KUKA KRL program: EPS_2_251806_MH49A_A_20260213065148.src

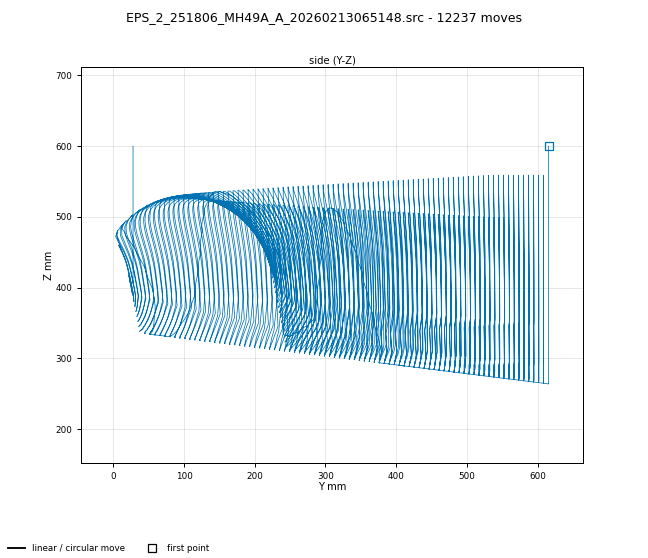
[picture p0: tool path of EPS_2_251806_MH49A_A_20260213065148.src, 12237 of 12239 moves have a stored position in this frame; points joined in program order, loops and branches not executed]
&ACCESS RVP
&REL 4
&COMMENT QRS 19112012
&PARAM EDITMASK = *
DEF PART()
EXT BAS (BAS_COMMAND :IN,REAL :IN )
INT I
BAS (#INITMOV,0 )

;KUKA QRS Post kuka4.cps  Date:22-06-2017 !

File_ID=3036

QRS_PRE_INIT()

;Init var - Until changes are made in qrs_pre_init
Outlet_Square_prg=0
Inlet_1_Square_prg=0
Inlet_2_Square_prg=0
Inlet_3_Square_prg=0
Inlet_4_Square_prg=0
Inlet_5_Square_prg=0

Outlet_1={X 0.000, Y 535.490, Z 458.500, B 0.000, E1 0.000 }
Inlet_1={X 0.000, Y 539.770, Z 398.500, B 0.000, E1 242.000 }
Outlet_1_type=201
Inlet_1_type=201
;QRS#1=Sidecore dimensions
;QRS#2=200-8" PVC SDR 35
;QRS#3=200-8" PVC SDR 35
;QRS#4=
;QRS#5=
;QRS#6=
;QRS#7=
;QRS#8=
;QRS#9=12-08 PSX
;QRS#10=12-08 PSX
;QRS#11=
;QRS#12=
;QRS#13=
;QRS#14=
;QRS#15=
;QRS#16=1220x127x838 2,75'
;QRS#17=EPS Height
;QRS#18=559
;QRS#19=*
;QRS#20= UPDATED VERSION 22-06-2017
;QRS#21=*
Outlet_Square=0100
Inlet_1_Square=0100
Inlet_2_Square=0
Inlet_3_Square=0
Inlet_4_Square=0
Inlet_5_Square=0
Mill_Square=1
Outlet_Square_Prg=204
Inlet_1_Square_prg=204

QRS_INIT()

$ADVANCE=5

; T1
PTP {E1 173.582,E2 173.582}
PTP {X 0,Y 615.48,A -85,B 0,C 180,E1 173.582,E2 173.582,E3 0,E4 0,E5 0,E6 0}
QRS_SPEED_INIT()
LIN {X 0,Y 615.48,Z 600,A -85,B 0,C 180,E1 173.582,E2 173.582,E3 0,E4 0,E5 0,E6 0} C_VEL
LIN {X 0,Y 615.48,Z 273.871,A -85,B 0,C 180,E1 173.582,E2 173.582} C_VEL
LIN {X 0,Y 615.48,Z 265.699,A -85,B 0,C 180,E1 173.582,E2 173.582} C_VEL
LIN {X 0,Y 615.469,Z 263.699,A -85,B 0,C 180,E1 173.396,E2 173.396} C_VEL
LIN {X 0,Y 615.482,Z 263.691,A -85,B 0,C 180,E1 170.801,E2 170.801} C_VEL
LIN {X 0,Y 615.433,Z 263.694,A -85,B 0,C 180,E1 168.138,E2 168.138} C_VEL
LIN {X 0,Y 615.433,Z 263.694,A -85,B 0,C 180,E1 166.069,E2 166.069} C_VEL
LIN {X 0,Y 615.451,Z 263.697,A -85,B 0,C 180,E1 163.565,E2 163.565} C_VEL
LIN {X 0,Y 615.479,Z 263.689,A -85,B 0,C 180,E1 160.662,E2 160.662} C_VEL
LIN {X 0,Y 615.473,Z 263.689,A -85,B 0,C 180,E1 158.568,E2 158.568} C_VEL
LIN {X 0,Y 615.439,Z 263.693,A -85,B 0,C 180,E1 155.991,E2 155.991} C_VEL
LIN {X 0,Y 615.452,Z 263.696,A -85,B 0,C 180,E1 153.555,E2 153.555} C_VEL
LIN {X 0,Y 615.483,Z 263.688,A -85,B 0,C 180,E1 150.594,E2 150.594} C_VEL
LIN {X 0,Y 615.462,Z 263.688,A -85,B 0,C 180,E1 148.314,E2 148.314} C_VEL
LIN {X 0,Y 615.443,Z 263.692,A -85,B 0,C 180,E1 145.976,E2 145.976} C_VEL
LIN {X 0,Y 615.453,Z 263.695,A -85,B 0,C 180,E1 143.573,E2 143.573} C_VEL
LIN {X 0,Y 615.495,Z 263.696,A -85,B 0,C 180,E1 140.932,E2 140.932} C_VEL
LIN {X 0,Y 615.496,Z 263.684,A -85,B 0,C 180,E1 138.527,E2 138.527} C_VEL
LIN {X 0,Y 615.449,Z 263.691,A -85,B 0,C 180,E1 135.847,E2 135.847} C_VEL
LIN {X 0,Y 615.487,Z 263.703,A -85,B 0,C 180,E1 133.048,E2 133.048} C_VEL
LIN {X 0,Y 615.465,Z 263.687,A -85,B 0,C 180,E1 130.087,E2 130.087} C_VEL
LIN {X 0,Y 615.462,Z 263.687,A -85,B 0,C 180,E1 128.01,E2 128.01} C_VEL
LIN {X 0,Y 615.456,Z 263.692,A -85,B 0,C 180,E1 125.615,E2 125.615} C_VEL
LIN {X 0,Y 615.472,Z 263.698,A -85,B 0,C 180,E1 123.235,E2 123.235} C_VEL
LIN {X 0,Y 615.488,Z 263.699,A -85,B 0,C 180,E1 120.917,E2 120.917} C_VEL
LIN {X 0,Y 615.466,Z 263.687,A -85,B 0,C 180,E1 117.914,E2 117.914} C_VEL
LIN {X 0,Y 615.461,Z 263.692,A -85,B 0,C 180,E1 115.565,E2 115.565} C_VEL
LIN {X 0,Y 615.487,Z 263.698,A -85,B 0,C 180,E1 112.843,E2 112.843} C_VEL
LIN {X 0,Y 615.481,Z 263.683,A -85,B 0,C 180,E1 110.032,E2 110.032} C_VEL
LIN {X 0,Y 615.473,Z 263.695,A -85,B 0,C 180,E1 107.27,E2 107.27} C_VEL
LIN {X 0,Y 615.485,Z 263.69,A -85,B 0,C 180,E1 104.549,E2 104.549} C_VEL
LIN {X 0,Y 615.477,Z 263.684,A -85,B 0,C 180,E1 101.861,E2 101.861} C_VEL
LIN {X 0,Y 615.477,Z 263.696,A -85,B 0,C 180,E1 99.199,E2 99.199} C_VEL
LIN {X 0,Y 615.483,Z 263.691,A -85,B 0,C 180,E1 96.557,E2 96.557} C_VEL
LIN {X 0,Y 615.485,Z 263.682,A -85,B 0,C 180,E1 93.929,E2 93.929} C_VEL
LIN {X 0,Y 615.474,Z 263.693,A -85,B 0,C 180,E1 91.31,E2 91.31} C_VEL
LIN {X 0,Y 615.485,Z 263.696,A -85,B 0,C 180,E1 88.693,E2 88.693} C_VEL
LIN {X 0,Y 615.487,Z 263.682,A -85,B 0,C 180,E1 86.073,E2 86.073} C_VEL
LIN {X 0,Y 615.475,Z 263.689,A -85,B 0,C 180,E1 83.429,E2 83.429} C_VEL
LIN {X 0,Y 615.49,Z 263.699,A -85,B 0,C 180,E1 80.803,E2 80.803} C_VEL
LIN {X 0,Y 615.481,Z 263.685,A -85,B 0,C 180,E1 78.141,E2 78.141} C_VEL
LIN {X 0,Y 615.478,Z 263.687,A -85,B 0,C 180,E1 75.453,E2 75.453} C_VEL
LIN {X 0,Y 615.488,Z 263.698,A -85,B 0,C 180,E1 72.732,E2 72.732} C_VEL
LIN {X 0,Y 615.484,Z 263.683,A -85,B 0,C 180,E1 69.97,E2 69.97} C_VEL
LIN {X 0,Y 615.482,Z 263.693,A -85,B 0,C 180,E1 67.159,E2 67.159} C_VEL
LIN {X 0,Y 615.474,Z 263.693,A -85,B 0,C 180,E1 64.433,E2 64.433} C_VEL
LIN {X 0,Y 615.473,Z 263.687,A -85,B 0,C 180,E1 62.088,E2 62.088} C_VEL
LIN {X 0,Y 615.483,Z 263.683,A -85,B 0,C 180,E1 59.844,E2 59.844} C_VEL
LIN {X 0,Y 615.494,Z 263.682,A -85,B 0,C 180,E1 57.548,E2 57.548} C_VEL
LIN {X 0,Y 615.484,Z 263.69,A -85,B 0,C 180,E1 55.19,E2 55.19} C_VEL
LIN {X 0,Y 615.491,Z 263.701,A -85,B 0,C 180,E1 52.764,E2 52.764} C_VEL
LIN {X 0,Y 615.47,Z 263.686,A -85,B 0,C 180,E1 49.912,E2 49.912} C_VEL
LIN {X 0,Y 615.487,Z 263.682,A -85,B 0,C 180,E1 47.654,E2 47.654} C_VEL
LIN {X 0,Y 615.489,Z 263.799,A -85,B 0,C 180,E1 45.291,E2 45.291} C_VEL
LIN {X 0,Y 615.45,Z 278.087,A -85,B 0,C 180,E1 42.705,E2 42.705} C_VEL
LIN {X 0,Y 615.463,Z 288.652,A -85,B 0,C 180,E1 40.808,E2 40.808} C_VEL
LIN {X 0,Y 615.487,Z 395.253,A -85,B 0,C 180,E1 39.537,E2 39.537} C_VEL
LIN {X 0,Y 615.489,Z 408.573,A -85,B 0,C 180,E1 39.239,E2 39.239} C_VEL
LIN {X 0,Y 615.487,Z 421.763,A -85,B 0,C 180,E1 38.799,E2 38.799} C_VEL
LIN {X 0,Y 615.467,Z 433.203,A -85,B 0,C 180,E1 38.278,E2 38.278} C_VEL
LIN {X 0,Y 615.479,Z 444.346,A -85,B 0,C 180,E1 37.629,E2 37.629} C_VEL
LIN {X 0,Y 615.495,Z 455.472,A -85,B 0,C 180,E1 36.816,E2 36.816} C_VEL
LIN {X 0,Y 615.497,Z 464.537,A -85,B 0,C 180,E1 35.989,E2 35.989} C_VEL
LIN {X 0,Y 615.496,Z 473.253,A -85,B 0,C 180,E1 35.014,E2 35.014} C_VEL
LIN {X 0,Y 615.496,Z 480.397,A -85,B 0,C 180,E1 34.021,E2 34.021} C_VEL
LIN {X 0,Y 615.496,Z 484.99,A -85,B 0,C 180,E1 33.235,E2 33.235} C_VEL
LIN {X 0,Y 615.493,Z 490.657,A -85,B 0,C 180,E1 32.013,E2 32.013} C_VEL
LIN {X 0,Y 615.497,Z 494.308,A -85,B 0,C 180,E1 30.919,E2 30.919} C_VEL
LIN {X 0,Y 615.496,Z 496.791,A -85,B 0,C 180,E1 29.808,E2 29.808} C_VEL
LIN {X 0,Y 615.497,Z 498.269,A -85,B 0,C 180,E1 28.465,E2 28.465} C_VEL
LIN {X 0,Y 615.496,Z 498.086,A -85,B 0,C 180,E1 27.176,E2 27.176} C_VEL
LIN {X 0,Y 615.494,Z 497.341,A -85,B 0,C 180,E1 26.443,E2 26.443} C_VEL
LIN {X 0,Y 615.495,Z 495.782,A -85,B 0,C 180,E1 25.585,E2 25.585} C_VEL
LIN {X 0,Y 615.495,Z 493.234,A -85,B 0,C 180,E1 24.631,E2 24.631} C_VEL
LIN {X 0,Y 615.496,Z 489.236,A -85,B 0,C 180,E1 23.556,E2 23.556} C_VEL
LIN {X 0,Y 615.496,Z 484.603,A -85,B 0,C 180,E1 22.604,E2 22.604} C_VEL
LIN {X 0,Y 615.495,Z 478.501,A -85,B 0,C 180,E1 21.607,E2 21.607} C_VEL
LIN {X 0,Y 615.497,Z 470.633,A -85,B 0,C 180,E1 20.578,E2 20.578} C_VEL
LIN {X 0,Y 615.497,Z 462.118,A -85,B 0,C 180,E1 19.684,E2 19.684} C_VEL
LIN {X 0,Y 615.498,Z 451.961,A -85,B 0,C 180,E1 18.818,E2 18.818} C_VEL
LIN {X 0,Y 615.464,Z 441.937,A -85,B 0,C 180,E1 18.125,E2 18.125} C_VEL
LIN {X 0,Y 615.471,Z 431.12,A -85,B 0,C 180,E1 17.528,E2 17.528} C_VEL
LIN {X 0,Y 615.474,Z 418.019,A -85,B 0,C 180,E1 16.971,E2 16.971} C_VEL
LIN {X 0,Y 615.451,Z 405.553,A -85,B 0,C 180,E1 16.587,E2 16.587} C_VEL
LIN {X 0,Y 615.45,Z 392.084,A -85,B 0,C 180,E1 16.325,E2 16.325} C_VEL
LIN {X 0,Y 615.493,Z 288.624,A -85,B 0,C 180,E1 15.098,E2 15.098} C_VEL
LIN {X 0,Y 615.482,Z 274.331,A -85,B 0,C 180,E1 12.53,E2 12.53} C_VEL
LIN {X 0,Y 615.427,Z 263.699,A -85,B 0,C 180,E1 10.576,E2 10.576} C_VEL
LIN {X 0,Y 615.425,Z 263.699,A -85,B 0,C 180,E1 8.537,E2 8.537} C_VEL
LIN {X 0,Y 615.426,Z 263.699,A -85,B 0,C 180,E1 6.557,E2 6.557} C_VEL
LIN {X 0,Y 615.435,Z 263.698,A -85,B 0,C 180,E1 4.585,E2 4.585} C_VEL
LIN {X 0,Y 615.44,Z 263.698,A -85,B 0,C 180,E1 2.618,E2 2.618} C_VEL
LIN {X 0,Y 615.412,Z 263.699,A -85,B 0,C 180,E1 0,E2 0} C_VEL
LIN {X 0,Y 615.451,Z 263.699,A -85,B 0,C 180,E1 -2.618,E2 -2.618} C_VEL
LIN {X 0,Y 615.468,Z 263.697,A -85,B 0,C 180,E1 -5.242,E2 -5.242} C_VEL
LIN {X 0,Y 615.417,Z 263.698,A -85,B 0,C 180,E1 -7.877,E2 -7.877} C_VEL
LIN {X 0,Y 615.419,Z 263.697,A -85,B 0,C 180,E1 -9.864,E2 -9.864} C_VEL
LIN {X 0,Y 615.42,Z 263.697,A -85,B 0,C 180,E1 -11.862,E2 -11.862} C_VEL
LIN {X 0,Y 615.419,Z 263.697,A -85,B 0,C 180,E1 -13.935,E2 -13.935} C_VEL
LIN {X 0,Y 615.421,Z 263.697,A -85,B 0,C 180,E1 -15.907,E2 -15.907} C_VEL
LIN {X 0,Y 615.421,Z 263.697,A -85,B 0,C 180,E1 -17.959,E2 -17.959} C_VEL
LIN {X 0,Y 615.418,Z 263.697,A -85,B 0,C 180,E1 -20.035,E2 -20.035} C_VEL
LIN {X 0,Y 615.422,Z 263.698,A -85,B 0,C 180,E1 -22.348,E2 -22.348} C_VEL
LIN {X 0,Y 615.481,Z 263.7,A -85,B 0,C 180,E1 -24.992,E2 -24.992} C_VEL
LIN {X 0,Y 615.486,Z 263.701,A -85,B 0,C 180,E1 -27.178,E2 -27.178} C_VEL
LIN {X 0,Y 615.423,Z 263.696,A -85,B 0,C 180,E1 -30.164,E2 -30.164} C_VEL
LIN {X 0,Y 615.427,Z 263.697,A -85,B 0,C 180,E1 -32.461,E2 -32.461} C_VEL
LIN {X 0,Y 615.45,Z 263.699,A -85,B 0,C 180,E1 -34.818,E2 -34.818} C_VEL
LIN {X 0,Y 615.496,Z 263.699,A -85,B 0,C 180,E1 -37.242,E2 -37.242} C_VEL
LIN {X 0,Y 615.431,Z 263.695,A -85,B 0,C 180,E1 -40.091,E2 -40.091} C_VEL
LIN {X 0,Y 615.425,Z 263.696,A -85,B 0,C 180,E1 -42.359,E2 -42.359} C_VEL
LIN {X 0,Y 615.431,Z 263.694,A -85,B 0,C 180,E1 -44.155,E2 -44.155} C_VEL
LIN {X 0,Y 615.457,Z 263.698,A -85,B 0,C 180,E1 -46.956,E2 -46.956} C_VEL
LIN {X 0,Y 615.453,Z 263.692,A -85,B 0,C 180,E1 -49.915,E2 -49.915} C_VEL
LIN {X 0,Y 615.448,Z 263.693,A -85,B 0,C 180,E1 -51.993,E2 -51.993} C_VEL
LIN {X 0,Y 615.43,Z 263.694,A -85,B 0,C 180,E1 -54.386,E2 -54.386} C_VEL
LIN {X 0,Y 615.434,Z 263.697,A -85,B 0,C 180,E1 -56.766,E2 -56.766} C_VEL
LIN {X 0,Y 615.463,Z 263.698,A -85,B 0,C 180,E1 -59.084,E2 -59.084} C_VEL
LIN {X 0,Y 615.451,Z 263.692,A -85,B 0,C 180,E1 -62.087,E2 -62.087} C_VEL
LIN {X 0,Y 615.434,Z 263.694,A -85,B 0,C 180,E1 -64.442,E2 -64.442} C_VEL
LIN {X 0,Y 615.435,Z 263.73,A -85,B 0,C 180,E1 -66.69,E2 -66.69} C_VEL
LIN {X 0,Y 615.481,Z 283.686,A -85,B 0,C 180,E1 -69.272,E2 -69.272} C_VEL
LIN {X 0,Y 615.476,Z 305.498,A -85,B 0,C 180,E1 -72.046,E2 -72.046} C_VEL
LIN {X 0,Y 615.49,Z 327.283,A -85,B 0,C 180,E1 -74.777,E2 -74.777} C_VEL
LIN {X 0,Y 615.45,Z 346.155,A -85,B 0,C 180,E1 -77.115,E2 -77.115} C_VEL
LIN {X 0,Y 615.457,Z 454.961,A -85,B 0,C 180,E1 -78.412,E2 -78.412} C_VEL
LIN {X 0,Y 615.456,Z 467.431,A -85,B 0,C 180,E1 -78.683,E2 -78.683} C_VEL
LIN {X 0,Y 615.483,Z 480.691,A -85,B 0,C 180,E1 -79.116,E2 -79.116} C_VEL
LIN {X 0,Y 615.49,Z 492.517,A -85,B 0,C 180,E1 -79.642,E2 -79.642} C_VEL
LIN {X 0,Y 615.488,Z 504.026,A -85,B 0,C 180,E1 -80.306,E2 -80.306} C_VEL
LIN {X 0,Y 615.499,Z 514.366,A -85,B 0,C 180,E1 -81.052,E2 -81.052} C_VEL
LIN {X 0,Y 615.497,Z 522.832,A -85,B 0,C 180,E1 -81.796,E2 -81.796} C_VEL
LIN {X 0,Y 615.497,Z 531.98,A -85,B 0,C 180,E1 -82.786,E2 -82.786} C_VEL
LIN {X 0,Y 615.498,Z 539.326,A -85,B 0,C 180,E1 -83.774,E2 -83.774} C_VEL
LIN {X 0,Y 615.498,Z 545.213,A -85,B 0,C 180,E1 -84.76,E2 -84.76} C_VEL
LIN {X 0,Y 615.494,Z 549.858,A -85,B 0,C 180,E1 -85.745,E2 -85.745} C_VEL
LIN {X 0,Y 615.494,Z 553.403,A -85,B 0,C 180,E1 -86.728,E2 -86.728} C_VEL
LIN {X 0,Y 615.497,Z 555.236,A -85,B 0,C 180,E1 -87.383,E2 -87.383} C_VEL
LIN {X 0,Y 615.498,Z 556.61,A -85,B 0,C 180,E1 -88.038,E2 -88.038} C_VEL
LIN {X 0,Y 615.496,Z 558.174,A -85,B 0,C 180,E1 -89.347,E2 -89.347} C_VEL
LIN {X 0,Y 615.494,Z 558.389,A -85,B 0,C 180,E1 -90.001,E2 -90.001} C_VEL
LIN {X 0,Y 615.495,Z 557.579,A -85,B 0,C 180,E1 -91.309,E2 -91.309} C_VEL
LIN {X 0,Y 615.498,Z 556.606,A -85,B 0,C 180,E1 -91.964,E2 -91.964} C_VEL
LIN {X 0,Y 615.497,Z 555.231,A -85,B 0,C 180,E1 -92.619,E2 -92.619} C_VEL
LIN {X 0,Y 615.496,Z 552.347,A -85,B 0,C 180,E1 -93.601,E2 -93.601} C_VEL
LIN {X 0,Y 615.498,Z 548.439,A -85,B 0,C 180,E1 -94.585,E2 -94.585} C_VEL
LIN {X 0,Y 615.499,Z 543.402,A -85,B 0,C 180,E1 -95.57,E2 -95.57} C_VEL
LIN {X 0,Y 615.497,Z 536.87,A -85,B 0,C 180,E1 -96.583,E2 -96.583} C_VEL
LIN {X 0,Y 615.497,Z 529.13,A -85,B 0,C 180,E1 -97.546,E2 -97.546} C_VEL
LIN {X 0,Y 615.498,Z 521.043,A -85,B 0,C 180,E1 -98.371,E2 -98.371} C_VEL
LIN {X 0,Y 615.499,Z 511.166,A -85,B 0,C 180,E1 -99.199,E2 -99.199} C_VEL
LIN {X 0,Y 615.489,Z 499.98,A -85,B 0,C 180,E1 -99.945,E2 -99.945} C_VEL
LIN {X 0,Y 615.489,Z 489.022,A -85,B 0,C 180,E1 -100.527,E2 -100.527} C_VEL
LIN {X 0,Y 615.469,Z 476.532,A -85,B 0,C 180,E1 -101.039,E2 -101.039} C_VEL
LIN {X 0,Y 615.454,Z 464.076,A -85,B 0,C 180,E1 -101.402,E2 -101.402} C_VEL
LIN {X 0,Y 615.459,Z 450.483,A -85,B 0,C 180,E1 -101.652,E2 -101.652} C_VEL
LIN {X 0,Y 615.449,Z 346.138,A -85,B 0,C 180,E1 -102.887,E2 -102.887} C_VEL
LIN {X 0,Y 615.48,Z 325.904,A -85,B 0,C 180,E1 -105.395,E2 -105.395} C_VEL
LIN {X 0,Y 615.485,Z 304.214,A -85,B 0,C 180,E1 -108.116,E2 -108.116} C_VEL
LIN {X 0,Y 615.485,Z 282.304,A -85,B 0,C 180,E1 -110.905,E2 -110.905} C_VEL
LIN {X 0,Y 615.435,Z 263.712,A -85,B 0,C 180,E1 -113.312,E2 -113.312} C_VEL
LIN {X 0,Y 615.44,Z 263.693,A -85,B 0,C 180,E1 -115.716,E2 -115.716} C_VEL
LIN {X 0,Y 615.48,Z 263.702,A -85,B 0,C 180,E1 -118.656,E2 -118.656} C_VEL
LIN {X 0,Y 615.444,Z 263.698,A -85,B 0,C 180,E1 -121.079,E2 -121.079} C_VEL
LIN {X 0,Y 615.434,Z 263.697,A -85,B 0,C 180,E1 -123.237,E2 -123.237} C_VEL
LIN {X 0,Y 615.427,Z 263.695,A -85,B 0,C 180,E1 -125.617,E2 -125.617} C_VEL
LIN {X 0,Y 615.452,Z 263.694,A -85,B 0,C 180,E1 -128.068,E2 -128.068} C_VEL
LIN {X 0,Y 615.442,Z 263.698,A -85,B 0,C 180,E1 -131.089,E2 -131.089} C_VEL
LIN {X 0,Y 615.43,Z 263.698,A -85,B 0,C 180,E1 -133.246,E2 -133.246} C_VEL
LIN {X 0,Y 615.436,Z 263.696,A -85,B 0,C 180,E1 -136.003,E2 -136.003} C_VEL
LIN {X 0,Y 615.464,Z 263.699,A -85,B 0,C 180,E1 -138.903,E2 -138.903} C_VEL
LIN {X 0,Y 615.44,Z 263.7,A -85,B 0,C 180,E1 -141.092,E2 -141.092} C_VEL
LIN {X 0,Y 615.414,Z 263.699,A -85,B 0,C 180,E1 -143.57,E2 -143.57} C_VEL
LIN {X 0,Y 615.468,Z 263.699,A -85,B 0,C 180,E1 -146.462,E2 -146.462} C_VEL
LIN {X 0,Y 615.444,Z 263.7,A -85,B 0,C 180,E1 -149.078,E2 -149.078} C_VEL
LIN {X 0,Y 615.41,Z 263.7,A -85,B 0,C 180,E1 -151.555,E2 -151.555} C_VEL
LIN {X 0,Y 615.409,Z 263.7,A -85,B 0,C 180,E1 -153.552,E2 -153.552} C_VEL
LIN {X 0,Y 615.414,Z 263.7,A -85,B 0,C 180,E1 -155.997,E2 -155.997} C_VEL
LIN {X 0,Y 615.471,Z 263.7,A -85,B 0,C 180,E1 -158.567,E2 -158.567} C_VEL
LIN {X 0,Y 615.424,Z 263.699,A -85,B 0,C 180,E1 -161.399,E2 -161.399} C_VEL
LIN {X 0,Y 615.416,Z 263.698,A -85,B 0,C 180,E1 -163.575,E2 -163.575} C_VEL
LIN {X 0,Y 615.424,Z 263.698,A -85,B 0,C 180,E1 -165.449,E2 -165.449} C_VEL
LIN {X 0,Y 615.426,Z 263.697,A -85,B 0,C 180,E1 -167.468,E2 -167.468} C_VEL
LIN {X 0,Y 615.428,Z 263.697,A -85,B 0,C 180,E1 -169.472,E2 -169.472} C_VEL
LIN {X 0,Y 615.431,Z 263.696,A -85,B 0,C 180,E1 -171.462,E2 -171.462} C_VEL
LIN {X 0,Y 615.432,Z 263.697,A -85,B 0,C 180,E1 -173.442,E2 -173.442} C_VEL
LIN {X 0,Y 615.44,Z 263.695,A -85,B 0,C 180,E1 -175.415,E2 -175.415} C_VEL
LIN {X 0,Y 615.446,Z 263.695,A -85,B 0,C 180,E1 -177.382,E2 -177.382} C_VEL
LIN {X 0,Y 615.452,Z 263.694,A -85,B 0,C 180,E1 -179.345,E2 -179.345} C_VEL
LIN {X 0,Y 615.425,Z 263.696,A -85,B 0,C 180,E1 -181.963,E2 -181.963} C_VEL
LIN {X 0,Y 615.467,Z 263.699,A -85,B 0,C 180,E1 -184.584,E2 -184.584} C_VEL
LIN {X 0,Y 615.469,Z 263.699,A -85,B 0,C 180,E1 -186.604,E2 -186.604} C_VEL
LIN {X 0,Y 614.804,Z 263.839,A -85,B 0,C 180,E1 -187.15,E2 -187.15} C_VEL
LIN {X 0,Y 611.979,Z 264.248,A -85,B 0,C 180,E1 -188.036,E2 -188.036} C_VEL
LIN {X 0,Y 609.581,Z 264.561,A -85,B 0,C 180,E1 -188.749,E2 -188.749} C_VEL
LIN {X 0,Y 608.531,Z 264.681,A -85,B 0,C 180,E1 -189.298,E2 -189.298} C_VEL
LIN {X 0,Y 608.434,Z 264.691,A -85,B 0,C 180,E1 -189.484,E2 -189.484} C_VEL
LIN {X 0,Y 608.415,Z 264.692,A -85,B 0,C 180,E1 -192,E2 -192} C_VEL
LIN {X 0,Y 608.454,Z 264.696,A -85,B 0,C 180,E1 -194.721,E2 -194.721} C_VEL
LIN {X 0,Y 608.433,Z 264.691,A -85,B 0,C 180,E1 -197.477,E2 -197.477} C_VEL
LIN {X 0,Y 608.427,Z 264.691,A -85,B 0,C 180,E1 -199.571,E2 -199.571} C_VEL
LIN {X 0,Y 608.434,Z 264.693,A -85,B 0,C 180,E1 -202.406,E2 -202.406} C_VEL
LIN {X 0,Y 608.443,Z 264.692,A -85,B 0,C 180,E1 -205.301,E2 -205.301} C_VEL
LIN {X 0,Y 608.428,Z 264.692,A -85,B 0,C 180,E1 -207.519,E2 -207.519} C_VEL
LIN {X 0,Y 608.43,Z 264.69,A -85,B 0,C 180,E1 -209.973,E2 -209.973} C_VEL
LIN {X 0,Y 608.43,Z 264.694,A -85,B 0,C 180,E1 -212.525,E2 -212.525} C_VEL
LIN {X 0,Y 608.436,Z 264.694,A -85,B 0,C 180,E1 -215.278,E2 -215.278} C_VEL
LIN {X 0,Y 608.445,Z 264.688,A -85,B 0,C 180,E1 -217.748,E2 -217.748} C_VEL
LIN {X 0,Y 608.422,Z 264.693,A -85,B 0,C 180,E1 -220.331,E2 -220.331} C_VEL
LIN {X 0,Y 608.456,Z 264.698,A -85,B 0,C 180,E1 -222.959,E2 -222.959} C_VEL
LIN {X 0,Y 608.437,Z 264.689,A -85,B 0,C 180,E1 -225.737,E2 -225.737} C_VEL
LIN {X 0,Y 608.442,Z 264.688,A -85,B 0,C 180,E1 -227.941,E2 -227.941} C_VEL
LIN {X 0,Y 608.465,Z 264.692,A -85,B 0,C 180,E1 -230.702,E2 -230.702} C_VEL
LIN {X 0,Y 608.465,Z 264.695,A -85,B 0,C 180,E1 -233.089,E2 -233.089} C_VEL
LIN {X 0,Y 608.466,Z 264.688,A -85,B 0,C 180,E1 -235.533,E2 -235.533} C_VEL
LIN {X 0,Y 608.461,Z 264.686,A -85,B 0,C 180,E1 -237.908,E2 -237.908} C_VEL
LIN {X 0,Y 608.446,Z 264.688,A -85,B 0,C 180,E1 -240.221,E2 -240.221} C_VEL
LIN {X 0,Y 608.475,Z 264.691,A -85,B 0,C 180,E1 -242.793,E2 -242.793} C_VEL
LIN {X 0,Y 608.472,Z 264.685,A -85,B 0,C 180,E1 -245.848,E2 -245.848} C_VEL
LIN {X 0,Y 608.456,Z 264.688,A -85,B 0,C 180,E1 -248.309,E2 -248.309} C_VEL
LIN {X 0,Y 608.451,Z 264.697,A -85,B 0,C 180,E1 -251.131,E2 -251.131} C_VEL
LIN {X 0,Y 608.455,Z 264.687,A -85,B 0,C 180,E1 -253.907,E2 -253.907} C_VEL
LIN {X 0,Y 608.451,Z 264.691,A -85,B 0,C 180,E1 -256.644,E2 -256.644} C_VEL
LIN {X 0,Y 608.463,Z 264.691,A -85,B 0,C 180,E1 -259.35,E2 -259.35} C_VEL
LIN {X 0,Y 608.474,Z 264.684,A -85,B 0,C 180,E1 -262.033,E2 -262.033} C_VEL
LIN {X 0,Y 608.456,Z 264.691,A -85,B 0,C 180,E1 -264.698,E2 -264.698} C_VEL
LIN {X 0,Y 608.474,Z 264.69,A -85,B 0,C 180,E1 -267.351,E2 -267.351} C_VEL
LIN {X 0,Y 608.477,Z 264.684,A -85,B 0,C 180,E1 -269.999,E2 -269.999} C_VEL
LIN {X 0,Y 608.466,Z 264.689,A -85,B 0,C 180,E1 -272.647,E2 -272.647} C_VEL
LIN {X 0,Y 608.466,Z 264.693,A -85,B 0,C 180,E1 -275.3,E2 -275.3} C_VEL
LIN {X 0,Y 608.474,Z 264.684,A -85,B 0,C 180,E1 -277.965,E2 -277.965} C_VEL
LIN {X 0,Y 608.458,Z 264.689,A -85,B 0,C 180,E1 -280.648,E2 -280.648} C_VEL
LIN {X 0,Y 608.465,Z 264.692,A -85,B 0,C 180,E1 -283.354,E2 -283.354} C_VEL
LIN {X 0,Y 608.456,Z 264.687,A -85,B 0,C 180,E1 -286.091,E2 -286.091} C_VEL
LIN {X 0,Y 608.447,Z 264.694,A -85,B 0,C 180,E1 -288.867,E2 -288.867} C_VEL
LIN {X 0,Y 608.464,Z 264.688,A -85,B 0,C 180,E1 -291.688,E2 -291.688} C_VEL
LIN {X 0,Y 608.451,Z 264.689,A -85,B 0,C 180,E1 -294.567,E2 -294.567} C_VEL
LIN {X 0,Y 608.476,Z 264.695,A -85,B 0,C 180,E1 -297.208,E2 -297.208} C_VEL
LIN {X 0,Y 608.454,Z 264.687,A -85,B 0,C 180,E1 -299.97,E2 -299.97} C_VEL
LIN {X 0,Y 608.463,Z 264.687,A -85,B 0,C 180,E1 -302.523,E2 -302.523} C_VEL
LIN {X 0,Y 608.434,Z 264.699,A -85,B 0,C 180,E1 -305.273,E2 -305.273} C_VEL
LIN {X 0,Y 608.457,Z 264.689,A -85,B 0,C 180,E1 -307.741,E2 -307.741} C_VEL
LIN {X 0,Y 608.447,Z 264.688,A -85,B 0,C 180,E1 -310.329,E2 -310.329} C_VEL
LIN {X 0,Y 608.48,Z 264.694,A -85,B 0,C 180,E1 -313.31,E2 -313.31} C_VEL
LIN {X 0,Y 608.502,Z 264.835,A -85,B 0,C 180,E1 -314.674,E2 -314.674} C_VEL
LIN {X 0,Y 608.432,Z 279.669,A -85,B 0,C 180,E1 -317.38,E2 -317.38} C_VEL
LIN {X 0,Y 608.439,Z 288.884,A -85,B 0,C 180,E1 -319.046,E2 -319.046} C_VEL
LIN {X 0,Y 608.552,Z 395.169,A -85,B 0,C 180,E1 -320.326,E2 -320.326} C_VEL
LIN {X 0,Y 608.547,Z 408.611,A -85,B 0,C 180,E1 -320.628,E2 -320.628} C_VEL
LIN {X 0,Y 608.517,Z 421.099,A -85,B 0,C 180,E1 -321.045,E2 -321.045} C_VEL
LIN {X 0,Y 608.487,Z 431.65,A -85,B 0,C 180,E1 -321.515,E2 -321.515} C_VEL
LIN {X 0,Y 608.464,Z 442.542,A -85,B 0,C 180,E1 -322.128,E2 -322.128} C_VEL
LIN {X 0,Y 608.491,Z 452.552,A -85,B 0,C 180,E1 -322.83,E2 -322.83} C_VEL
LIN {X 0,Y 608.474,Z 462.7,A -85,B 0,C 180,E1 -323.705,E2 -323.705} C_VEL
LIN {X 0,Y 608.449,Z 470.445,A -85,B 0,C 180,E1 -324.52,E2 -324.52} C_VEL
LIN {X 0,Y 608.459,Z 478.293,A -85,B 0,C 180,E1 -325.53,E2 -325.53} C_VEL
LIN {X 0,Y 608.432,Z 484.497,A -85,B 0,C 180,E1 -326.526,E2 -326.526} C_VEL
LIN {X 0,Y 608.43,Z 489.222,A -85,B 0,C 180,E1 -327.471,E2 -327.471} C_VEL
LIN {X 0,Y 608.447,Z 493.912,A -85,B 0,C 180,E1 -328.721,E2 -328.721} C_VEL
LIN {X 0,Y 608.446,Z 495.945,A -85,B 0,C 180,E1 -329.454,E2 -329.454} C_VEL
LIN {X 0,Y 608.442,Z 497.468,A -85,B 0,C 180,E1 -330.22,E2 -330.22} C_VEL
LIN {X 0,Y 608.423,Z 498.778,A -85,B 0,C 180,E1 -331.376,E2 -331.376} C_VEL
LIN {X 0,Y 608.427,Z 498.726,A -85,B 0,C 180,E1 -332.789,E2 -332.789} C_VEL
LIN {X 0,Y 608.416,Z 497.313,A -85,B 0,C 180,E1 -333.964,E2 -333.964} C_VEL
LIN {X 0,Y 608.428,Z 494.822,A -85,B 0,C 180,E1 -335.064,E2 -335.064} C_VEL
LIN {X 0,Y 608.437,Z 491.173,A -85,B 0,C 180,E1 -336.154,E2 -336.154} C_VEL
LIN {X 0,Y 608.456,Z 486.303,A -85,B 0,C 180,E1 -337.231,E2 -337.231} C_VEL
LIN {X 0,Y 608.458,Z 479.982,A -85,B 0,C 180,E1 -338.308,E2 -338.308} C_VEL
LIN {X 0,Y 608.462,Z 472.656,A -85,B 0,C 180,E1 -339.305,E2 -339.305} C_VEL
LIN {X 0,Y 608.471,Z 464.052,A -85,B 0,C 180,E1 -340.255,E2 -340.255} C_VEL
LIN {X 0,Y 608.495,Z 454.173,A -85,B 0,C 180,E1 -341.132,E2 -341.132} C_VEL
LIN {X 0,Y 608.476,Z 443.243,A -85,B 0,C 180,E1 -341.916,E2 -341.916} C_VEL
LIN {X 0,Y 608.492,Z 432.647,A -85,B 0,C 180,E1 -342.525,E2 -342.525} C_VEL
LIN {X 0,Y 608.523,Z 421.091,A -85,B 0,C 180,E1 -343.045,E2 -343.045} C_VEL
LIN {X 0,Y 608.499,Z 407.986,A -85,B 0,C 180,E1 -343.48,E2 -343.48} C_VEL
LIN {X 0,Y 608.509,Z 394.771,A -85,B 0,C 180,E1 -343.772,E2 -343.772} C_VEL
LIN {X 0,Y 608.452,Z 288.885,A -85,B 0,C 180,E1 -345.044,E2 -345.044} C_VEL
LIN {X 0,Y 608.442,Z 274.43,A -85,B 0,C 180,E1 -347.662,E2 -347.662} C_VEL
LIN {X 0,Y 608.405,Z 264.695,A -85,B 0,C 180,E1 -349.476,E2 -349.476} C_VEL
LIN {X 0,Y 608.405,Z 264.693,A -85,B 0,C 180,E1 -352.032,E2 -352.032} C_VEL
LIN {X 0,Y 608.443,Z 264.696,A -85,B 0,C 180,E1 -354.698,E2 -354.698} C_VEL
LIN {X 0,Y 608.431,Z 264.693,A -85,B 0,C 180,E1 -357.352,E2 -357.352} C_VEL
LIN {X 0,Y 608.403,Z 264.693,A -85,B 0,C 180,E1 -360,E2 -360} C_VEL
LIN {X 0,Y 608.439,Z 264.694,A -85,B 0,C 180,E1 -362.649,E2 -362.649} C_VEL
LIN {X 0,Y 608.44,Z 264.694,A -85,B 0,C 180,E1 -365.302,E2 -365.302} C_VEL
LIN {X 0,Y 608.411,Z 264.692,A -85,B 0,C 180,E1 -367.968,E2 -367.968} C_VEL
LIN {X 0,Y 608.427,Z 264.695,A -85,B 0,C 180,E1 -370.651,E2 -370.651} C_VEL
LIN {X 0,Y 608.444,Z 264.693,A -85,B 0,C 180,E1 -373.357,E2 -373.357} C_VEL
LIN {X 0,Y 608.398,Z 264.694,A -85,B 0,C 180,E1 -376.096,E2 -376.096} C_VEL
LIN {X 0,Y 608.435,Z 264.697,A -85,B 0,C 180,E1 -378.871,E2 -378.871} C_VEL
LIN {X 0,Y 608.43,Z 264.691,A -85,B 0,C 180,E1 -381.693,E2 -381.693} C_VEL
LIN {X 0,Y 608.411,Z 264.694,A -85,B 0,C 180,E1 -384.573,E2 -384.573} C_VEL
LIN {X 0,Y 608.469,Z 264.694,A -85,B 0,C 180,E1 -387.219,E2 -387.219} C_VEL
LIN {X 0,Y 608.415,Z 264.692,A -85,B 0,C 180,E1 -389.975,E2 -389.975} C_VEL
LIN {X 0,Y 608.405,Z 264.694,A -85,B 0,C 180,E1 -392.525,E2 -392.525} C_VEL
LIN {X 0,Y 608.441,Z 264.694,A -85,B 0,C 180,E1 -394.914,E2 -394.914} C_VEL
LIN {X 0,Y 608.435,Z 264.691,A -85,B 0,C 180,E1 -397.749,E2 -397.749} C_VEL
LIN {X 0,Y 608.397,Z 264.694,A -85,B 0,C 180,E1 -400.331,E2 -400.331} C_VEL
LIN {X 0,Y 608.396,Z 264.694,A -85,B 0,C 180,E1 -402.335,E2 -402.335} C_VEL
LIN {X 0,Y 608.405,Z 264.693,A -85,B 0,C 180,E1 -404.266,E2 -404.266} C_VEL
LIN {X 0,Y 608.427,Z 264.697,A -85,B 0,C 180,E1 -407.045,E2 -407.045} C_VEL
LIN {X 0,Y 608.434,Z 264.693,A -85,B 0,C 180,E1 -409.702,E2 -409.702} C_VEL
LIN {X 0,Y 608.429,Z 264.69,A -85,B 0,C 180,E1 -412.257,E2 -412.257} C_VEL
LIN {X 0,Y 608.438,Z 264.696,A -85,B 0,C 180,E1 -415.097,E2 -415.097} C_VEL
LIN {X 0,Y 608.452,Z 264.689,A -85,B 0,C 180,E1 -417.91,E2 -417.91} C_VEL
LIN {X 0,Y 608.427,Z 264.69,A -85,B 0,C 180,E1 -420.223,E2 -420.223} C_VEL
LIN {X 0,Y 608.414,Z 264.692,A -85,B 0,C 180,E1 -422.485,E2 -422.485} C_VEL
LIN {X 0,Y 608.44,Z 264.7,A -85,B 0,C 180,E1 -425.432,E2 -425.432} C_VEL
LIN {X 0,Y 608.414,Z 264.753,A -85,B 0,C 180,E1 -426.54,E2 -426.54} C_VEL
LIN {X 0,Y 608.587,Z 275.5,A -85,B 0,C 180,E1 -427.96,E2 -427.96} C_VEL
LIN {X 0,Y 608.538,Z 295.969,A -85,B 0,C 180,E1 -430.611,E2 -430.611} C_VEL
LIN {X 0,Y 608.52,Z 316.438,A -85,B 0,C 180,E1 -433.221,E2 -433.221} C_VEL
LIN {X 0,Y 608.499,Z 339.388,A -85,B 0,C 180,E1 -436.105,E2 -436.105} C_VEL
LIN {X 0,Y 608.462,Z 346.452,A -85,B 0,C 180,E1 -436.975,E2 -436.975} C_VEL
LIN {X 0,Y 608.52,Z 455.07,A -85,B 0,C 180,E1 -438.278,E2 -438.278} C_VEL
LIN {X 0,Y 608.491,Z 468.297,A -85,B 0,C 180,E1 -438.573,E2 -438.573} C_VEL
LIN {X 0,Y 608.509,Z 480.68,A -85,B 0,C 180,E1 -438.984,E2 -438.984} C_VEL
LIN {X 0,Y 608.507,Z 492.675,A -85,B 0,C 180,E1 -439.521,E2 -439.521} C_VEL
LIN {X 0,Y 608.477,Z 504.229,A -85,B 0,C 180,E1 -440.193,E2 -440.193} C_VEL
LIN {X 0,Y 608.485,Z 514.619,A -85,B 0,C 180,E1 -440.948,E2 -440.948} C_VEL
LIN {X 0,Y 608.474,Z 523.132,A -85,B 0,C 180,E1 -441.701,E2 -441.701} C_VEL
LIN {X 0,Y 608.47,Z 530.976,A -85,B 0,C 180,E1 -442.536,E2 -442.536} C_VEL
LIN {X 0,Y 608.46,Z 538.293,A -85,B 0,C 180,E1 -443.485,E2 -443.485} C_VEL
LIN {X 0,Y 608.45,Z 543.875,A -85,B 0,C 180,E1 -444.367,E2 -444.367} C_VEL
LIN {X 0,Y 608.432,Z 548.957,A -85,B 0,C 180,E1 -445.364,E2 -445.364} C_VEL
LIN {X 0,Y 608.449,Z 552.901,A -85,B 0,C 180,E1 -446.359,E2 -446.359} C_VEL
LIN {X 0,Y 608.425,Z 555.812,A -85,B 0,C 180,E1 -447.353,E2 -447.353} C_VEL
LIN {X 0,Y 608.443,Z 557.203,A -85,B 0,C 180,E1 -448.015,E2 -448.015} C_VEL
LIN {X 0,Y 608.438,Z 558.784,A -85,B 0,C 180,E1 -449.339,E2 -449.339} C_VEL
LIN {X 0,Y 608.434,Z 559,A -85,B 0,C 180,E1 -450.001,E2 -450.001} C_VEL
LIN {X 0,Y 608.448,Z 558.183,A -85,B 0,C 180,E1 -451.325,E2 -451.325} C_VEL
LIN {X 0,Y 608.443,Z 557.2,A -85,B 0,C 180,E1 -451.987,E2 -451.987} C_VEL
LIN {X 0,Y 608.425,Z 555.807,A -85,B 0,C 180,E1 -452.649,E2 -452.649} C_VEL
LIN {X 0,Y 608.449,Z 552.894,A -85,B 0,C 180,E1 -453.643,E2 -453.643} C_VEL
LIN {X 0,Y 608.432,Z 548.947,A -85,B 0,C 180,E1 -454.638,E2 -454.638} C_VEL
LIN {X 0,Y 608.437,Z 542.874,A -85,B 0,C 180,E1 -455.801,E2 -455.801} C_VEL
LIN {X 0,Y 608.462,Z 536.232,A -85,B 0,C 180,E1 -456.8,E2 -456.8} C_VEL
LIN {X 0,Y 608.456,Z 527.987,A -85,B 0,C 180,E1 -457.8,E2 -457.8} C_VEL
LIN {X 0,Y 608.472,Z 519.534,A -85,B 0,C 180,E1 -458.636,E2 -458.636} C_VEL
LIN {X 0,Y 608.477,Z 509.089,A -85,B 0,C 180,E1 -459.473,E2 -459.473} C_VEL
LIN {X 0,Y 608.488,Z 498.755,A -85,B 0,C 180,E1 -460.145,E2 -460.145} C_VEL
LIN {X 0,Y 608.517,Z 487.606,A -85,B 0,C 180,E1 -460.724,E2 -460.724} C_VEL
LIN {X 0,Y 608.512,Z 475.907,A -85,B 0,C 180,E1 -461.192,E2 -461.192} C_VEL
LIN {X 0,Y 608.52,Z 463.271,A -85,B 0,C 180,E1 -461.555,E2 -461.555} C_VEL
LIN {X 0,Y 608.522,Z 450.61,A -85,B 0,C 180,E1 -461.787,E2 -461.787} C_VEL
LIN {X 0,Y 608.434,Z 346.271,A -85,B 0,C 180,E1 -463.038,E2 -463.038} C_VEL
LIN {X 0,Y 608.508,Z 327.337,A -85,B 0,C 180,E1 -465.404,E2 -465.404} C_VEL
LIN {X 0,Y 608.554,Z 304.236,A -85,B 0,C 180,E1 -468.33,E2 -468.33} C_VEL
LIN {X 0,Y 608.594,Z 282.305,A -85,B 0,C 180,E1 -471.153,E2 -471.153} C_VEL
LIN {X 0,Y 608.532,Z 265.248,A -85,B 0,C 180,E1 -473.389,E2 -473.389} C_VEL
LIN {X 0,Y 608.428,Z 264.692,A -85,B 0,C 180,E1 -473.484,E2 -473.484} C_VEL
LIN {X 0,Y 608.425,Z 264.693,A -85,B 0,C 180,E1 -476.035,E2 -476.035} C_VEL
LIN {X 0,Y 608.473,Z 264.695,A -85,B 0,C 180,E1 -478.619,E2 -478.619} C_VEL
LIN {X 0,Y 608.422,Z 264.692,A -85,B 0,C 180,E1 -481.317,E2 -481.317} C_VEL
LIN {X 0,Y 608.413,Z 264.692,A -85,B 0,C 180,E1 -483.726,E2 -483.726} C_VEL
LIN {X 0,Y 608.428,Z 264.692,A -85,B 0,C 180,E1 -486.091,E2 -486.091} C_VEL
LIN {X 0,Y 608.415,Z 264.702,A -85,B 0,C 180,E1 -488.589,E2 -488.589} C_VEL
LIN {X 0,Y 608.41,Z 264.693,A -85,B 0,C 180,E1 -491.336,E2 -491.336} C_VEL
LIN {X 0,Y 608.422,Z 264.691,A -85,B 0,C 180,E1 -493.87,E2 -493.87} C_VEL
LIN {X 0,Y 608.466,Z 264.696,A -85,B 0,C 180,E1 -496.687,E2 -496.687} C_VEL
LIN {X 0,Y 608.44,Z 264.697,A -85,B 0,C 180,E1 -498.822,E2 -498.822} C_VEL
LIN {X 0,Y 608.412,Z 264.692,A -85,B 0,C 180,E1 -501.761,E2 -501.761} C_VEL
LIN {X 0,Y 608.408,Z 264.693,A -85,B 0,C 180,E1 -503.953,E2 -503.953} C_VEL
LIN {X 0,Y 608.435,Z 264.694,A -85,B 0,C 180,E1 -506.327,E2 -506.327} C_VEL
LIN {X 0,Y 608.448,Z 264.698,A -85,B 0,C 180,E1 -508.725,E2 -508.725} C_VEL
LIN {X 0,Y 608.408,Z 264.694,A -85,B 0,C 180,E1 -511.383,E2 -511.383} C_VEL
LIN {X 0,Y 608.4,Z 264.696,A -85,B 0,C 180,E1 -513.223,E2 -513.223} C_VEL
LIN {X 0,Y 608.385,Z 264.696,A -85,B 0,C 180,E1 -515.857,E2 -515.857} C_VEL
LIN {X 0,Y 608.43,Z 264.694,A -85,B 0,C 180,E1 -518.307,E2 -518.307} C_VEL
LIN {X 0,Y 608.418,Z 264.694,A -85,B 0,C 180,E1 -521.285,E2 -521.285} C_VEL
LIN {X 0,Y 608.396,Z 264.694,A -85,B 0,C 180,E1 -523.904,E2 -523.904} C_VEL
LIN {X 0,Y 608.453,Z 264.696,A -85,B 0,C 180,E1 -526.643,E2 -526.643} C_VEL
LIN {X 0,Y 608.419,Z 264.693,A -85,B 0,C 180,E1 -529.349,E2 -529.349} C_VEL
LIN {X 0,Y 608.412,Z 264.694,A -85,B 0,C 180,E1 -531.363,E2 -531.363} C_VEL
LIN {X 0,Y 608.431,Z 264.692,A -85,B 0,C 180,E1 -533.367,E2 -533.367} C_VEL
LIN {X 0,Y 608.412,Z 264.694,A -85,B 0,C 180,E1 -535.362,E2 -535.362} C_VEL
LIN {X 0,Y 608.438,Z 264.691,A -85,B 0,C 180,E1 -537.351,E2 -537.351} C_VEL
LIN {X 0,Y 608.417,Z 264.692,A -85,B 0,C 180,E1 -540,E2 -540} C_VEL
LIN {X 0,Y 608.458,Z 264.694,A -85,B 0,C 180,E1 -542.648,E2 -542.648} C_VEL
LIN {X 0,Y 608.445,Z 264.691,A -85,B 0,C 180,E1 -545.302,E2 -545.302} C_VEL
LIN {X 0,Y 608.426,Z 264.69,A -85,B 0,C 180,E1 -547.967,E2 -547.967} C_VEL
LIN {X 0,Y 608.434,Z 264.691,A -85,B 0,C 180,E1 -549.484,E2 -549.484} C_VEL
LIN {X 0,Y 607.733,Z 264.779,A -85,B 0,C 180,E1 -550.037,E2 -550.037} C_VEL
LIN {X 0,Y 604.865,Z 265.143,A -85,B 0,C 180,E1 -550.934,E2 -550.934} C_VEL
LIN {X 0,Y 602.469,Z 265.437,A -85,B 0,C 180,E1 -551.656,E2 -551.656} C_VEL
LIN {X 0,Y 601.452,Z 265.561,A -85,B 0,C 180,E1 -552.213,E2 -552.213} C_VEL
LIN {X 0,Y 601.375,Z 265.572,A -85,B 0,C 180,E1 -552.401,E2 -552.401} C_VEL
LIN {X 0,Y 601.407,Z 265.575,A -85,B 0,C 180,E1 -554.897,E2 -554.897} C_VEL
LIN {X 0,Y 601.371,Z 265.57,A -85,B 0,C 180,E1 -557.689,E2 -557.689} C_VEL
LIN {X 0,Y 601.402,Z 265.57,A -85,B 0,C 180,E1 -560.522,E2 -560.522} C_VEL
LIN {X 0,Y 601.395,Z 265.569,A -85,B 0,C 180,E1 -563.411,E2 -563.411} C_VEL
LIN {X 0,Y 601.378,Z 265.571,A -85,B 0,C 180,E1 -566.364,E2 -566.364} C_VEL
LIN {X 0,Y 601.416,Z 265.573,A -85,B 0,C 180,E1 -568.793,E2 -568.793} C_VEL
LIN {X 0,Y 601.414,Z 265.566,A -85,B 0,C 180,E1 -571.461,E2 -571.461} C_VEL
LIN {X 0,Y 601.404,Z 265.566,A -85,B 0,C 180,E1 -574.119,E2 -574.119} C_VEL
LIN {X 0,Y 601.397,Z 265.571,A -85,B 0,C 180,E1 -576.583,E2 -576.583} C_VEL
LIN {X 0,Y 601.422,Z 265.565,A -85,B 0,C 180,E1 -579.539,E2 -579.539} C_VEL
LIN {X 0,Y 601.403,Z 265.566,A -85,B 0,C 180,E1 -581.766,E2 -581.766} C_VEL
LIN {X 0,Y 601.4,Z 265.57,A -85,B 0,C 180,E1 -584.537,E2 -584.537} C_VEL
LIN {X 0,Y 601.424,Z 265.566,A -85,B 0,C 180,E1 -587.408,E2 -587.408} C_VEL
LIN {X 0,Y 601.398,Z 265.566,A -85,B 0,C 180,E1 -590.007,E2 -590.007} C_VEL
LIN {X 0,Y 601.422,Z 265.568,A -85,B 0,C 180,E1 -592.619,E2 -592.619} C_VEL
LIN {X 0,Y 601.432,Z 265.571,A -85,B 0,C 180,E1 -595.072,E2 -595.072} C_VEL
LIN {X 0,Y 601.434,Z 265.564,A -85,B 0,C 180,E1 -597.487,E2 -597.487} C_VEL
LIN {X 0,Y 601.416,Z 265.564,A -85,B 0,C 180,E1 -599.853,E2 -599.853} C_VEL
LIN {X 0,Y 601.413,Z 265.564,A -85,B 0,C 180,E1 -602.134,E2 -602.134} C_VEL
LIN {X 0,Y 601.398,Z 265.575,A -85,B 0,C 180,E1 -605.123,E2 -605.123} C_VEL
LIN {X 0,Y 601.41,Z 265.569,A -85,B 0,C 180,E1 -607.395,E2 -607.395} C_VEL
LIN {X 0,Y 601.398,Z 265.566,A -85,B 0,C 180,E1 -610.191,E2 -610.191} C_VEL
LIN {X 0,Y 601.426,Z 265.573,A -85,B 0,C 180,E1 -613.015,E2 -613.015} C_VEL
LIN {X 0,Y 601.418,Z 265.564,A -85,B 0,C 180,E1 -615.908,E2 -615.908} C_VEL
LIN {X 0,Y 601.43,Z 265.565,A -85,B 0,C 180,E1 -618.542,E2 -618.542} C_VEL
LIN {X 0,Y 601.432,Z 265.569,A -85,B 0,C 180,E1 -621.262,E2 -621.262} C_VEL
LIN {X 0,Y 601.411,Z 265.564,A -85,B 0,C 180,E1 -623.962,E2 -623.962} C_VEL
LIN {X 0,Y 601.418,Z 265.567,A -85,B 0,C 180,E1 -626.65,E2 -626.65} C_VEL
LIN {X 0,Y 601.45,Z 265.566,A -85,B 0,C 180,E1 -629.329,E2 -629.329} C_VEL
LIN {X 0,Y 601.433,Z 265.562,A -85,B 0,C 180,E1 -632.008,E2 -632.008} C_VEL
LIN {X 0,Y 601.413,Z 265.568,A -85,B 0,C 180,E1 -634.691,E2 -634.691} C_VEL
LIN {X 0,Y 601.452,Z 265.565,A -85,B 0,C 180,E1 -637.383,E2 -637.383} C_VEL
LIN {X 0,Y 601.426,Z 265.562,A -85,B 0,C 180,E1 -640.093,E2 -640.093} C_VEL
LIN {X 0,Y 601.417,Z 265.569,A -85,B 0,C 180,E1 -642.826,E2 -642.826} C_VEL
LIN {X 0,Y 601.415,Z 265.567,A -85,B 0,C 180,E1 -645.589,E2 -645.589} C_VEL
LIN {X 0,Y 601.411,Z 265.565,A -85,B 0,C 180,E1 -648.389,E2 -648.389} C_VEL
LIN {X 0,Y 601.399,Z 265.575,A -85,B 0,C 180,E1 -651.236,E2 -651.236} C_VEL
LIN {X 0,Y 601.412,Z 265.571,A -85,B 0,C 180,E1 -653.407,E2 -653.407} C_VEL
LIN {X 0,Y 601.399,Z 265.566,A -85,B 0,C 180,E1 -656.36,E2 -656.36} C_VEL
LIN {X 0,Y 601.433,Z 265.566,A -85,B 0,C 180,E1 -658.789,E2 -658.789} C_VEL
LIN {X 0,Y 601.425,Z 265.569,A -85,B 0,C 180,E1 -661.456,E2 -661.456} C_VEL
LIN {X 0,Y 601.414,Z 265.564,A -85,B 0,C 180,E1 -664.114,E2 -664.114} C_VEL
LIN {X 0,Y 601.401,Z 265.567,A -85,B 0,C 180,E1 -666.577,E2 -666.577} C_VEL
LIN {X 0,Y 601.421,Z 265.569,A -85,B 0,C 180,E1 -669.534,E2 -669.534} C_VEL
LIN {X 0,Y 601.426,Z 265.564,A -85,B 0,C 180,E1 -672.593,E2 -672.593} C_VEL
LIN {X 0,Y 601.459,Z 265.634,A -85,B 0,C 180,E1 -674.613,E2 -674.613} C_VEL
LIN {X 0,Y 601.405,Z 280.743,A -85,B 0,C 180,E1 -677.402,E2 -677.402} C_VEL
LIN {X 0,Y 601.41,Z 288.842,A -85,B 0,C 180,E1 -678.883,E2 -678.883} C_VEL
LIN {X 0,Y 601.67,Z 295.653,A -85,B 0,C 180,E1 -678.981,E2 -678.981} C_VEL
LIN {X 0,Y 601.61,Z 395.299,A -85,B 0,C 180,E1 -680.191,E2 -680.191} C_VEL
LIN {X 0,Y 601.59,Z 408.377,A -85,B 0,C 180,E1 -680.487,E2 -680.487} C_VEL
LIN {X 0,Y 601.541,Z 421.424,A -85,B 0,C 180,E1 -680.928,E2 -680.928} C_VEL
LIN {X 0,Y 601.498,Z 433.019,A -85,B 0,C 180,E1 -681.463,E2 -681.463} C_VEL
LIN {X 0,Y 601.455,Z 443.185,A -85,B 0,C 180,E1 -682.054,E2 -682.054} C_VEL
LIN {X 0,Y 601.47,Z 453.576,A -85,B 0,C 180,E1 -682.803,E2 -682.803} C_VEL
LIN {X 0,Y 601.42,Z 463.946,A -85,B 0,C 180,E1 -683.727,E2 -683.727} C_VEL
LIN {X 0,Y 601.389,Z 473.282,A -85,B 0,C 180,E1 -684.777,E2 -684.777} C_VEL
LIN {X 0,Y 601.377,Z 481.089,A -85,B 0,C 180,E1 -685.879,E2 -685.879} C_VEL
LIN {X 0,Y 601.343,Z 487.336,A -85,B 0,C 180,E1 -687.01,E2 -687.01} C_VEL
LIN {X 0,Y 601.355,Z 492.587,A -85,B 0,C 180,E1 -688.271,E2 -688.271} C_VEL
LIN {X 0,Y 601.328,Z 494.99,A -85,B 0,C 180,E1 -689.053,E2 -689.053} C_VEL
LIN {X 0,Y 601.358,Z 496.858,A -85,B 0,C 180,E1 -689.851,E2 -689.851} C_VEL
LIN {X 0,Y 601.333,Z 498.063,A -85,B 0,C 180,E1 -690.603,E2 -690.603} C_VEL
LIN {X 0,Y 601.33,Z 498.779,A -85,B 0,C 180,E1 -691.368,E2 -691.368} C_VEL
LIN {X 0,Y 601.337,Z 498.835,A -85,B 0,C 180,E1 -692.638,E2 -692.638} C_VEL
LIN {X 0,Y 601.336,Z 497.876,A -85,B 0,C 180,E1 -693.634,E2 -693.634} C_VEL
LIN {X 0,Y 601.325,Z 496.561,A -85,B 0,C 180,E1 -694.378,E2 -694.378} C_VEL
LIN {X 0,Y 601.351,Z 494.77,A -85,B 0,C 180,E1 -695.12,E2 -695.12} C_VEL
LIN {X 0,Y 601.367,Z 491.101,A -85,B 0,C 180,E1 -696.223,E2 -696.223} C_VEL
LIN {X 0,Y 601.376,Z 485.796,A -85,B 0,C 180,E1 -697.387,E2 -697.387} C_VEL
LIN {X 0,Y 601.385,Z 479.859,A -85,B 0,C 180,E1 -698.401,E2 -698.401} C_VEL
LIN {X 0,Y 601.388,Z 471.959,A -85,B 0,C 180,E1 -699.477,E2 -699.477} C_VEL
LIN {X 0,Y 601.407,Z 463.887,A -85,B 0,C 180,E1 -700.369,E2 -700.369} C_VEL
LIN {X 0,Y 601.466,Z 454.148,A -85,B 0,C 180,E1 -701.241,E2 -701.241} C_VEL
LIN {X 0,Y 601.444,Z 444.307,A -85,B 0,C 180,E1 -701.962,E2 -701.962} C_VEL
LIN {X 0,Y 601.488,Z 433.929,A -85,B 0,C 180,E1 -702.578,E2 -702.578} C_VEL
LIN {X 0,Y 601.521,Z 422.322,A -85,B 0,C 180,E1 -703.125,E2 -703.125} C_VEL
LIN {X 0,Y 601.532,Z 408.969,A -85,B 0,C 180,E1 -703.587,E2 -703.587} C_VEL
LIN {X 0,Y 601.551,Z 395.794,A -85,B 0,C 180,E1 -703.891,E2 -703.891} C_VEL
LIN {X 0,Y 601.677,Z 315.43,A -85,B 0,C 180,E1 -704.872,E2 -704.872} C_VEL
LIN {X 0,Y 601.532,Z 289.844,A -85,B 0,C 180,E1 -705.182,E2 -705.182} C_VEL
LIN {X 0,Y 601.432,Z 288.693,A -85,B 0,C 180,E1 -705.233,E2 -705.233} C_VEL
LIN {X 0,Y 601.392,Z 274.387,A -85,B 0,C 180,E1 -707.857,E2 -707.857} C_VEL
LIN {X 0,Y 601.371,Z 265.572,A -85,B 0,C 180,E1 -709.521,E2 -709.521} C_VEL
LIN {X 0,Y 601.371,Z 265.569,A -85,B 0,C 180,E1 -711.939,E2 -711.939} C_VEL
LIN {X 0,Y 601.398,Z 265.572,A -85,B 0,C 180,E1 -714.636,E2 -714.636} C_VEL
LIN {X 0,Y 601.395,Z 265.57,A -85,B 0,C 180,E1 -717.321,E2 -717.321} C_VEL
LIN {X 0,Y 601.372,Z 265.569,A -85,B 0,C 180,E1 -720,E2 -720} C_VEL
LIN {X 0,Y 601.403,Z 265.571,A -85,B 0,C 180,E1 -722.68,E2 -722.68} C_VEL
LIN {X 0,Y 601.397,Z 265.57,A -85,B 0,C 180,E1 -725.365,E2 -725.365} C_VEL
LIN {X 0,Y 601.377,Z 265.568,A -85,B 0,C 180,E1 -728.062,E2 -728.062} C_VEL
LIN {X 0,Y 601.43,Z 265.572,A -85,B 0,C 180,E1 -731.05,E2 -731.05} C_VEL
LIN {X 0,Y 601.385,Z 265.57,A -85,B 0,C 180,E1 -733.517,E2 -733.517} C_VEL
LIN {X 0,Y 601.377,Z 265.569,A -85,B 0,C 180,E1 -736.289,E2 -736.289} C_VEL
LIN {X 0,Y 601.384,Z 265.578,A -85,B 0,C 180,E1 -739.1,E2 -739.1} C_VEL
LIN {X 0,Y 601.369,Z 265.569,A -85,B 0,C 180,E1 -741.961,E2 -741.961} C_VEL
LIN {X 0,Y 601.378,Z 265.569,A -85,B 0,C 180,E1 -744.296,E2 -744.296} C_VEL
LIN {X 0,Y 601.434,Z 265.572,A -85,B 0,C 180,E1 -747.112,E2 -747.112} C_VEL
LIN {X 0,Y 601.377,Z 265.568,A -85,B 0,C 180,E1 -750.152,E2 -750.152} C_VEL
LIN {X 0,Y 601.377,Z 265.572,A -85,B 0,C 180,E1 -752.72,E2 -752.72} C_VEL
LIN {X 0,Y 601.38,Z 265.578,A -85,B 0,C 180,E1 -755.12,E2 -755.12} C_VEL
LIN {X 0,Y 601.403,Z 265.572,A -85,B 0,C 180,E1 -757.422,E2 -757.422} C_VEL
LIN {X 0,Y 601.373,Z 265.569,A -85,B 0,C 180,E1 -759.998,E2 -759.998} C_VEL
LIN {X 0,Y 601.374,Z 265.571,A -85,B 0,C 180,E1 -762.674,E2 -762.674} C_VEL
LIN {X 0,Y 601.391,Z 265.574,A -85,B 0,C 180,E1 -765.486,E2 -765.486} C_VEL
LIN {X 0,Y 601.388,Z 265.567,A -85,B 0,C 180,E1 -768.238,E2 -768.238} C_VEL
LIN {X 0,Y 601.378,Z 265.572,A -85,B 0,C 180,E1 -770.877,E2 -770.877} C_VEL
LIN {X 0,Y 601.379,Z 265.578,A -85,B 0,C 180,E1 -773.421,E2 -773.421} C_VEL
LIN {X 0,Y 601.396,Z 265.567,A -85,B 0,C 180,E1 -776.07,E2 -776.07} C_VEL
LIN {X 0,Y 601.394,Z 265.567,A -85,B 0,C 180,E1 -778.55,E2 -778.55} C_VEL
LIN {X 0,Y 601.43,Z 265.573,A -85,B 0,C 180,E1 -781.377,E2 -781.377} C_VEL
LIN {X 0,Y 601.38,Z 265.569,A -85,B 0,C 180,E1 -784.14,E2 -784.14} C_VEL
LIN {X 0,Y 601.395,Z 265.606,A -85,B 0,C 180,E1 -786.364,E2 -786.364} C_VEL
LIN {X 0,Y 601.7,Z 270.044,A -85,B 0,C 180,E1 -786.969,E2 -786.969} C_VEL
LIN {X 0,Y 601.645,Z 290.51,A -85,B 0,C 180,E1 -789.668,E2 -789.668} C_VEL
LIN {X 0,Y 601.51,Z 312.344,A -85,B 0,C 180,E1 -792.494,E2 -792.494} C_VEL
LIN {X 0,Y 601.512,Z 331.449,A -85,B 0,C 180,E1 -794.935,E2 -794.935} C_VEL
LIN {X 0,Y 601.417,Z 346.452,A -85,B 0,C 180,E1 -796.82,E2 -796.82} C_VEL
LIN {X 0,Y 601.639,Z 370.597,A -85,B 0,C 180,E1 -797.115,E2 -797.115} C_VEL
LIN {X 0,Y 601.592,Z 455.07,A -85,B 0,C 180,E1 -798.141,E2 -798.141} C_VEL
LIN {X 0,Y 601.554,Z 468.298,A -85,B 0,C 180,E1 -798.44,E2 -798.44} C_VEL
LIN {X 0,Y 601.539,Z 479.955,A -85,B 0,C 180,E1 -798.827,E2 -798.827} C_VEL
LIN {X 0,Y 601.517,Z 492.674,A -85,B 0,C 180,E1 -799.398,E2 -799.398} C_VEL
LIN {X 0,Y 601.479,Z 504.23,A -85,B 0,C 180,E1 -800.078,E2 -800.078} C_VEL
LIN {X 0,Y 601.444,Z 514.62,A -85,B 0,C 180,E1 -800.841,E2 -800.841} C_VEL
LIN {X 0,Y 601.428,Z 523.132,A -85,B 0,C 180,E1 -801.603,E2 -801.603} C_VEL
LIN {X 0,Y 601.417,Z 530.976,A -85,B 0,C 180,E1 -802.448,E2 -802.448} C_VEL
LIN {X 0,Y 601.369,Z 538.233,A -85,B 0,C 180,E1 -803.399,E2 -803.399} C_VEL
LIN {X 0,Y 601.371,Z 543.875,A -85,B 0,C 180,E1 -804.301,E2 -804.301} C_VEL
LIN {X 0,Y 601.336,Z 548.957,A -85,B 0,C 180,E1 -805.309,E2 -805.309} C_VEL
LIN {X 0,Y 601.368,Z 552.901,A -85,B 0,C 180,E1 -806.316,E2 -806.316} C_VEL
LIN {X 0,Y 601.325,Z 555.812,A -85,B 0,C 180,E1 -807.322,E2 -807.322} C_VEL
LIN {X 0,Y 601.342,Z 557.204,A -85,B 0,C 180,E1 -807.992,E2 -807.992} C_VEL
LIN {X 0,Y 601.339,Z 558.785,A -85,B 0,C 180,E1 -809.331,E2 -809.331} C_VEL
LIN {X 0,Y 601.335,Z 559,A -85,B 0,C 180,E1 -810.001,E2 -810.001} C_VEL
LIN {X 0,Y 601.347,Z 558.183,A -85,B 0,C 180,E1 -811.34,E2 -811.34} C_VEL
LIN {X 0,Y 601.342,Z 557.201,A -85,B 0,C 180,E1 -812.01,E2 -812.01} C_VEL
LIN {X 0,Y 601.325,Z 555.807,A -85,B 0,C 180,E1 -812.68,E2 -812.68} C_VEL
LIN {X 0,Y 601.368,Z 552.894,A -85,B 0,C 180,E1 -813.686,E2 -813.686} C_VEL
LIN {X 0,Y 601.336,Z 548.947,A -85,B 0,C 180,E1 -814.693,E2 -814.693} C_VEL
LIN {X 0,Y 601.372,Z 542.874,A -85,B 0,C 180,E1 -815.87,E2 -815.87} C_VEL
LIN {X 0,Y 601.382,Z 536.233,A -85,B 0,C 180,E1 -816.88,E2 -816.88} C_VEL
LIN {X 0,Y 601.401,Z 527.987,A -85,B 0,C 180,E1 -817.893,E2 -817.893} C_VEL
LIN {X 0,Y 601.436,Z 519.535,A -85,B 0,C 180,E1 -818.738,E2 -818.738} C_VEL
LIN {X 0,Y 601.445,Z 509.091,A -85,B 0,C 180,E1 -819.585,E2 -819.585} C_VEL
LIN {X 0,Y 601.483,Z 498.757,A -85,B 0,C 180,E1 -820.264,E2 -820.264} C_VEL
LIN {X 0,Y 601.538,Z 486.595,A -85,B 0,C 180,E1 -820.896,E2 -820.896} C_VEL
LIN {X 0,Y 601.545,Z 474.219,A -85,B 0,C 180,E1 -821.379,E2 -821.379} C_VEL
LIN {X 0,Y 601.559,Z 461.442,A -85,B 0,C 180,E1 -821.733,E2 -821.733} C_VEL
LIN {X 0,Y 601.599,Z 449.094,A -85,B 0,C 180,E1 -821.946,E2 -821.946} C_VEL
LIN {X 0,Y 601.531,Z 347.163,A -85,B 0,C 180,E1 -823.169,E2 -823.169} C_VEL
LIN {X 0,Y 601.426,Z 346.271,A -85,B 0,C 180,E1 -823.193,E2 -823.193} C_VEL
LIN {X 0,Y 601.496,Z 327.337,A -85,B 0,C 180,E1 -825.589,E2 -825.589} C_VEL
LIN {X 0,Y 601.582,Z 305.504,A -85,B 0,C 180,E1 -828.386,E2 -828.386} C_VEL
LIN {X 0,Y 601.682,Z 283.67,A -85,B 0,C 180,E1 -831.228,E2 -831.228} C_VEL
LIN {X 0,Y 601.683,Z 267.295,A -85,B 0,C 180,E1 -833.398,E2 -833.398} C_VEL
LIN {X 0,Y 601.389,Z 265.572,A -85,B 0,C 180,E1 -833.661,E2 -833.661} C_VEL
LIN {X 0,Y 601.386,Z 265.575,A -85,B 0,C 180,E1 -836.363,E2 -836.363} C_VEL
LIN {X 0,Y 601.423,Z 265.57,A -85,B 0,C 180,E1 -838.786,E2 -838.786} C_VEL
LIN {X 0,Y 601.386,Z 265.568,A -85,B 0,C 180,E1 -841.726,E2 -841.726} C_VEL
LIN {X 0,Y 601.402,Z 265.568,A -85,B 0,C 180,E1 -844.117,E2 -844.117} C_VEL
LIN {X 0,Y 601.381,Z 265.578,A -85,B 0,C 180,E1 -846.582,E2 -846.582} C_VEL
LIN {X 0,Y 601.373,Z 265.572,A -85,B 0,C 180,E1 -849.126,E2 -849.126} C_VEL
LIN {X 0,Y 601.389,Z 265.567,A -85,B 0,C 180,E1 -851.764,E2 -851.764} C_VEL
LIN {X 0,Y 601.377,Z 265.577,A -85,B 0,C 180,E1 -854.53,E2 -854.53} C_VEL
LIN {X 0,Y 601.408,Z 265.571,A -85,B 0,C 180,E1 -856.425,E2 -856.425} C_VEL
LIN {X 0,Y 601.381,Z 265.569,A -85,B 0,C 180,E1 -859.425,E2 -859.425} C_VEL
LIN {X 0,Y 601.364,Z 265.57,A -85,B 0,C 180,E1 -861.727,E2 -861.727} C_VEL
LIN {X 0,Y 601.352,Z 265.575,A -85,B 0,C 180,E1 -864.243,E2 -864.243} C_VEL
LIN {X 0,Y 601.396,Z 265.577,A -85,B 0,C 180,E1 -866.684,E2 -866.684} C_VEL
LIN {X 0,Y 601.383,Z 265.572,A -85,B 0,C 180,E1 -869.056,E2 -869.056} C_VEL
LIN {X 0,Y 601.368,Z 265.571,A -85,B 0,C 180,E1 -871.37,E2 -871.37} C_VEL
LIN {X 0,Y 601.35,Z 265.572,A -85,B 0,C 180,E1 -873.633,E2 -873.633} C_VEL
LIN {X 0,Y 601.374,Z 265.577,A -85,B 0,C 180,E1 -876.587,E2 -876.587} C_VEL
LIN {X 0,Y 601.369,Z 265.57,A -85,B 0,C 180,E1 -879.476,E2 -879.476} C_VEL
LIN {X 0,Y 601.363,Z 265.574,A -85,B 0,C 180,E1 -882.31,E2 -882.31} C_VEL
LIN {X 0,Y 601.392,Z 265.571,A -85,B 0,C 180,E1 -885.102,E2 -885.102} C_VEL
LIN {X 0,Y 601.364,Z 265.57,A -85,B 0,C 180,E1 -887.856,E2 -887.856} C_VEL
LIN {X 0,Y 601.378,Z 265.569,A -85,B 0,C 180,E1 -889.904,E2 -889.904} C_VEL
LIN {X 0,Y 601.423,Z 265.571,A -85,B 0,C 180,E1 -892.614,E2 -892.614} C_VEL
LIN {X 0,Y 601.384,Z 265.57,A -85,B 0,C 180,E1 -895.307,E2 -895.307} C_VEL
LIN {X 0,Y 601.404,Z 265.568,A -85,B 0,C 180,E1 -897.32,E2 -897.32} C_VEL
LIN {X 0,Y 601.386,Z 265.568,A -85,B 0,C 180,E1 -900,E2 -900} C_VEL
LIN {X 0,Y 601.421,Z 265.572,A -85,B 0,C 180,E1 -902.679,E2 -902.679} C_VEL
LIN {X 0,Y 601.403,Z 265.568,A -85,B 0,C 180,E1 -905.364,E2 -905.364} C_VEL
LIN {X 0,Y 601.393,Z 265.567,A -85,B 0,C 180,E1 -908.061,E2 -908.061} C_VEL
LIN {X 0,Y 601.449,Z 265.567,A -85,B 0,C 180,E1 -911.047,E2 -911.047} C_VEL
LIN {X 0,Y 601.375,Z 265.572,A -85,B 0,C 180,E1 -912.401,E2 -912.401} C_VEL
LIN {X 0,Y 600.725,Z 265.66,A -85,B 0,C 180,E1 -912.961,E2 -912.961} C_VEL
LIN {X 0,Y 597.879,Z 266.017,A -85,B 0,C 180,E1 -913.868,E2 -913.868} C_VEL
LIN {X 0,Y 595.463,Z 266.315,A -85,B 0,C 180,E1 -914.599,E2 -914.599} C_VEL
LIN {X 0,Y 594.422,Z 266.441,A -85,B 0,C 180,E1 -915.162,E2 -915.162} C_VEL
LIN {X 0,Y 594.335,Z 266.449,A -85,B 0,C 180,E1 -915.353,E2 -915.353} C_VEL
LIN {X 0,Y 594.348,Z 266.444,A -85,B 0,C 180,E1 -917.905,E2 -917.905} C_VEL
LIN {X 0,Y 594.363,Z 266.453,A -85,B 0,C 180,E1 -920.924,E2 -920.924} C_VEL
LIN {X 0,Y 594.357,Z 266.444,A -85,B 0,C 180,E1 -923.705,E2 -923.705} C_VEL
LIN {X 0,Y 594.367,Z 266.45,A -85,B 0,C 180,E1 -926.7,E2 -926.7} C_VEL
LIN {X 0,Y 594.357,Z 266.452,A -85,B 0,C 180,E1 -928.999,E2 -928.999} C_VEL
LIN {X 0,Y 594.362,Z 266.443,A -85,B 0,C 180,E1 -931.648,E2 -931.648} C_VEL
LIN {X 0,Y 594.377,Z 266.446,A -85,B 0,C 180,E1 -934.58,E2 -934.58} C_VEL
LIN {X 0,Y 594.366,Z 266.45,A -85,B 0,C 180,E1 -937.088,E2 -937.088} C_VEL
LIN {X 0,Y 594.353,Z 266.444,A -85,B 0,C 180,E1 -939.777,E2 -939.777} C_VEL
LIN {X 0,Y 594.346,Z 266.447,A -85,B 0,C 180,E1 -942.377,E2 -942.377} C_VEL
LIN {X 0,Y 594.34,Z 266.452,A -85,B 0,C 180,E1 -945.193,E2 -945.193} C_VEL
LIN {X 0,Y 594.37,Z 266.443,A -85,B 0,C 180,E1 -947.629,E2 -947.629} C_VEL
LIN {X 0,Y 594.375,Z 266.442,A -85,B 0,C 180,E1 -950.323,E2 -950.323} C_VEL
LIN {X 0,Y 594.375,Z 266.451,A -85,B 0,C 180,E1 -952.916,E2 -952.916} C_VEL
LIN {X 0,Y 594.363,Z 266.443,A -85,B 0,C 180,E1 -955.863,E2 -955.863} C_VEL
LIN {X 0,Y 594.368,Z 266.447,A -85,B 0,C 180,E1 -958.652,E2 -958.652} C_VEL
LIN {X 0,Y 594.376,Z 266.451,A -85,B 0,C 180,E1 -961.043,E2 -961.043} C_VEL
LIN {X 0,Y 594.373,Z 266.441,A -85,B 0,C 180,E1 -963.979,E2 -963.979} C_VEL
LIN {X 0,Y 594.381,Z 266.441,A -85,B 0,C 180,E1 -966.297,E2 -966.297} C_VEL
LIN {X 0,Y 594.402,Z 266.445,A -85,B 0,C 180,E1 -969.225,E2 -969.225} C_VEL
LIN {X 0,Y 594.347,Z 266.444,A -85,B 0,C 180,E1 -972.096,E2 -972.096} C_VEL
LIN {X 0,Y 594.361,Z 266.443,A -85,B 0,C 180,E1 -974.219,E2 -974.219} C_VEL
LIN {X 0,Y 594.375,Z 266.442,A -85,B 0,C 180,E1 -976.321,E2 -976.321} C_VEL
LIN {X 0,Y 594.377,Z 266.451,A -85,B 0,C 180,E1 -979.095,E2 -979.095} C_VEL
LIN {X 0,Y 594.413,Z 266.437,A -85,B 0,C 180,E1 -981.843,E2 -981.843} C_VEL
LIN {X 0,Y 594.386,Z 266.442,A -85,B 0,C 180,E1 -984.572,E2 -984.572} C_VEL
LIN {X 0,Y 594.405,Z 266.444,A -85,B 0,C 180,E1 -987.288,E2 -987.288} C_VEL
LIN {X 0,Y 594.413,Z 266.436,A -85,B 0,C 180,E1 -989.999,E2 -989.999} C_VEL
LIN {X 0,Y 594.4,Z 266.442,A -85,B 0,C 180,E1 -992.709,E2 -992.709} C_VEL
LIN {X 0,Y 594.396,Z 266.444,A -85,B 0,C 180,E1 -995.426,E2 -995.426} C_VEL
LIN {X 0,Y 594.409,Z 266.437,A -85,B 0,C 180,E1 -998.155,E2 -998.155} C_VEL
LIN {X 0,Y 594.385,Z 266.45,A -85,B 0,C 180,E1 -1001.073,E2 -1001.073} C_VEL
LIN {X 0,Y 594.379,Z 266.443,A -85,B 0,C 180,E1 -1003.676,E2 -1003.676} C_VEL
LIN {X 0,Y 594.388,Z 266.443,A -85,B 0,C 180,E1 -1006.718,E2 -1006.718} C_VEL
LIN {X 0,Y 594.361,Z 266.45,A -85,B 0,C 180,E1 -1009.331,E2 -1009.331} C_VEL
LIN {X 0,Y 594.358,Z 266.448,A -85,B 0,C 180,E1 -1011.5,E2 -1011.5} C_VEL
LIN {X 0,Y 594.382,Z 266.442,A -85,B 0,C 180,E1 -1013.701,E2 -1013.701} C_VEL
LIN {X 0,Y 594.38,Z 266.443,A -85,B 0,C 180,E1 -1016.696,E2 -1016.696} C_VEL
LIN {X 0,Y 594.372,Z 266.448,A -85,B 0,C 180,E1 -1018.995,E2 -1018.995} C_VEL
LIN {X 0,Y 594.378,Z 266.444,A -85,B 0,C 180,E1 -1021.643,E2 -1021.643} C_VEL
LIN {X 0,Y 594.381,Z 266.442,A -85,B 0,C 180,E1 -1024.575,E2 -1024.575} C_VEL
LIN {X 0,Y 594.369,Z 266.45,A -85,B 0,C 180,E1 -1027.082,E2 -1027.082} C_VEL
LIN {X 0,Y 594.359,Z 266.445,A -85,B 0,C 180,E1 -1029.773,E2 -1029.773} C_VEL
LIN {X 0,Y 594.37,Z 266.442,A -85,B 0,C 180,E1 -1032.369,E2 -1032.369} C_VEL
LIN {X 0,Y 594.403,Z 266.496,A -85,B 0,C 180,E1 -1034.562,E2 -1034.562} C_VEL
LIN {X 0,Y 594.35,Z 280.297,A -85,B 0,C 180,E1 -1037.142,E2 -1037.142} C_VEL
LIN {X 0,Y 594.373,Z 289.13,A -85,B 0,C 180,E1 -1038.738,E2 -1038.738} C_VEL
LIN {X 0,Y 594.74,Z 294.42,A -85,B 0,C 180,E1 -1038.811,E2 -1038.811} C_VEL
LIN {X 0,Y 594.651,Z 395.106,A -85,B 0,C 180,E1 -1040.047,E2 -1040.047} C_VEL
LIN {X 0,Y 594.626,Z 408.992,A -85,B 0,C 180,E1 -1040.368,E2 -1040.368} C_VEL
LIN {X 0,Y 594.58,Z 422.211,A -85,B 0,C 180,E1 -1040.83,E2 -1040.83} C_VEL
LIN {X 0,Y 594.495,Z 432.928,A -85,B 0,C 180,E1 -1041.333,E2 -1041.333} C_VEL
LIN {X 0,Y 594.428,Z 443.482,A -85,B 0,C 180,E1 -1041.955,E2 -1041.955} C_VEL
LIN {X 0,Y 594.434,Z 453.965,A -85,B 0,C 180,E1 -1042.725,E2 -1042.725} C_VEL
LIN {X 0,Y 594.365,Z 463.975,A -85,B 0,C 180,E1 -1043.631,E2 -1043.631} C_VEL
LIN {X 0,Y 594.315,Z 473.132,A -85,B 0,C 180,E1 -1044.671,E2 -1044.671} C_VEL
LIN {X 0,Y 594.294,Z 480.19,A -85,B 0,C 180,E1 -1045.665,E2 -1045.665} C_VEL
LIN {X 0,Y 594.268,Z 485.785,A -85,B 0,C 180,E1 -1046.639,E2 -1046.639} C_VEL
LIN {X 0,Y 594.262,Z 491.213,A -85,B 0,C 180,E1 -1047.847,E2 -1047.847} C_VEL
LIN {X 0,Y 594.245,Z 495.048,A -85,B 0,C 180,E1 -1049.039,E2 -1049.039} C_VEL
LIN {X 0,Y 594.234,Z 497.536,A -85,B 0,C 180,E1 -1050.216,E2 -1050.216} C_VEL
LIN {X 0,Y 594.253,Z 498.569,A -85,B 0,C 180,E1 -1051.052,E2 -1051.052} C_VEL
LIN {X 0,Y 594.215,Z 498.942,A -85,B 0,C 180,E1 -1051.765,E2 -1051.765} C_VEL
LIN {X 0,Y 594.232,Z 498.877,A -85,B 0,C 180,E1 -1052.532,E2 -1052.532} C_VEL
LIN {X 0,Y 594.245,Z 498.304,A -85,B 0,C 180,E1 -1053.294,E2 -1053.294} C_VEL
LIN {X 0,Y 594.234,Z 497.25,A -85,B 0,C 180,E1 -1054.05,E2 -1054.05} C_VEL
LIN {X 0,Y 594.249,Z 494.723,A -85,B 0,C 180,E1 -1055.175,E2 -1055.175} C_VEL
LIN {X 0,Y 594.268,Z 491.027,A -85,B 0,C 180,E1 -1056.291,E2 -1056.291} C_VEL
LIN {X 0,Y 594.276,Z 485.465,A -85,B 0,C 180,E1 -1057.513,E2 -1057.513} C_VEL
LIN {X 0,Y 594.327,Z 478.64,A -85,B 0,C 180,E1 -1058.662,E2 -1058.662} C_VEL
LIN {X 0,Y 594.354,Z 470.303,A -85,B 0,C 180,E1 -1059.766,E2 -1059.766} C_VEL
LIN {X 0,Y 594.381,Z 461.843,A -85,B 0,C 180,E1 -1060.666,E2 -1060.666} C_VEL
LIN {X 0,Y 594.447,Z 452.61,A -85,B 0,C 180,E1 -1061.474,E2 -1061.474} C_VEL
LIN {X 0,Y 594.437,Z 442.686,A -85,B 0,C 180,E1 -1062.187,E2 -1062.187} C_VEL
LIN {X 0,Y 594.543,Z 430.641,A -85,B 0,C 180,E1 -1062.876,E2 -1062.876} C_VEL
LIN {X 0,Y 594.572,Z 417.286,A -85,B 0,C 180,E1 -1063.452,E2 -1063.452} C_VEL
LIN {X 0,Y 594.601,Z 405.052,A -85,B 0,C 180,E1 -1063.83,E2 -1063.83} C_VEL
LIN {X 0,Y 594.639,Z 393.292,A -85,B 0,C 180,E1 -1064.073,E2 -1064.073} C_VEL
LIN {X 0,Y 594.662,Z 290.865,A -85,B 0,C 180,E1 -1065.324,E2 -1065.324} C_VEL
LIN {X 0,Y 594.369,Z 288.829,A -85,B 0,C 180,E1 -1065.368,E2 -1065.368} C_VEL
LIN {X 0,Y 594.374,Z 274.338,A -85,B 0,C 180,E1 -1068.058,E2 -1068.058} C_VEL
LIN {X 0,Y 594.328,Z 266.45,A -85,B 0,C 180,E1 -1069.568,E2 -1069.568} C_VEL
LIN {X 0,Y 594.365,Z 266.447,A -85,B 0,C 180,E1 -1072.527,E2 -1072.527} C_VEL
LIN {X 0,Y 594.345,Z 266.45,A -85,B 0,C 180,E1 -1075.252,E2 -1075.252} C_VEL
LIN {X 0,Y 594.323,Z 266.448,A -85,B 0,C 180,E1 -1077.967,E2 -1077.967} C_VEL
LIN {X 0,Y 594.383,Z 266.446,A -85,B 0,C 180,E1 -1080.678,E2 -1080.678} C_VEL
LIN {X 0,Y 594.346,Z 266.448,A -85,B 0,C 180,E1 -1083.39,E2 -1083.39} C_VEL
LIN {X 0,Y 594.303,Z 266.45,A -85,B 0,C 180,E1 -1086.11,E2 -1086.11} C_VEL
LIN {X 0,Y 594.355,Z 266.444,A -85,B 0,C 180,E1 -1088.158,E2 -1088.158} C_VEL
LIN {X 0,Y 594.4,Z 266.447,A -85,B 0,C 180,E1 -1091.114,E2 -1091.114} C_VEL
LIN {X 0,Y 594.326,Z 266.447,A -85,B 0,C 180,E1 -1094.177,E2 -1094.177} C_VEL
LIN {X 0,Y 594.345,Z 266.453,A -85,B 0,C 180,E1 -1097.195,E2 -1097.195} C_VEL
LIN {X 0,Y 594.326,Z 266.446,A -85,B 0,C 180,E1 -1100.056,E2 -1100.056} C_VEL
LIN {X 0,Y 594.312,Z 266.453,A -85,B 0,C 180,E1 -1102.74,E2 -1102.74} C_VEL
LIN {X 0,Y 594.338,Z 266.455,A -85,B 0,C 180,E1 -1105.195,E2 -1105.195} C_VEL
LIN {X 0,Y 594.339,Z 266.449,A -85,B 0,C 180,E1 -1107.531,E2 -1107.531} C_VEL
LIN {X 0,Y 594.337,Z 266.446,A -85,B 0,C 180,E1 -1110.332,E2 -1110.332} C_VEL
LIN {X 0,Y 594.336,Z 266.452,A -85,B 0,C 180,E1 -1112.953,E2 -1112.953} C_VEL
LIN {X 0,Y 594.337,Z 266.452,A -85,B 0,C 180,E1 -1115.41,E2 -1115.41} C_VEL
LIN {X 0,Y 594.343,Z 266.445,A -85,B 0,C 180,E1 -1117.944,E2 -1117.944} C_VEL
LIN {X 0,Y 594.347,Z 266.448,A -85,B 0,C 180,E1 -1120.827,E2 -1120.827} C_VEL
LIN {X 0,Y 594.339,Z 266.447,A -85,B 0,C 180,E1 -1123.844,E2 -1123.844} C_VEL
LIN {X 0,Y 594.341,Z 266.447,A -85,B 0,C 180,E1 -1126.705,E2 -1126.705} C_VEL
LIN {X 0,Y 594.358,Z 266.451,A -85,B 0,C 180,E1 -1129.439,E2 -1129.439} C_VEL
LIN {X 0,Y 594.36,Z 266.443,A -85,B 0,C 180,E1 -1132.396,E2 -1132.396} C_VEL
LIN {X 0,Y 594.361,Z 266.453,A -85,B 0,C 180,E1 -1135.424,E2 -1135.424} C_VEL
LIN {X 0,Y 594.355,Z 266.444,A -85,B 0,C 180,E1 -1138.361,E2 -1138.361} C_VEL
LIN {X 0,Y 594.369,Z 266.447,A -85,B 0,C 180,E1 -1141.045,E2 -1141.045} C_VEL
LIN {X 0,Y 594.344,Z 266.447,A -85,B 0,C 180,E1 -1144.058,E2 -1144.058} C_VEL
LIN {X 0,Y 594.405,Z 266.63,A -85,B 0,C 180,E1 -1146.208,E2 -1146.208} C_VEL
LIN {X 0,Y 594.809,Z 271.406,A -85,B 0,C 180,E1 -1146.871,E2 -1146.871} C_VEL
LIN {X 0,Y 594.724,Z 291.875,A -85,B 0,C 180,E1 -1149.601,E2 -1149.601} C_VEL
LIN {X 0,Y 594.552,Z 313.709,A -85,B 0,C 180,E1 -1152.46,E2 -1152.46} C_VEL
LIN {X 0,Y 594.495,Z 332.813,A -85,B 0,C 180,E1 -1154.928,E2 -1154.928} C_VEL
LIN {X 0,Y 594.421,Z 346.452,A -85,B 0,C 180,E1 -1156.662,E2 -1156.662} C_VEL
LIN {X 0,Y 594.748,Z 352.712,A -85,B 0,C 180,E1 -1156.745,E2 -1156.745} C_VEL
LIN {X 0,Y 594.643,Z 455.07,A -85,B 0,C 180,E1 -1158.001,E2 -1158.001} C_VEL
LIN {X 0,Y 594.618,Z 468.299,A -85,B 0,C 180,E1 -1158.303,E2 -1158.303} C_VEL
LIN {X 0,Y 594.585,Z 481.328,A -85,B 0,C 180,E1 -1158.748,E2 -1158.748} C_VEL
LIN {X 0,Y 594.532,Z 492.673,A -85,B 0,C 180,E1 -1159.272,E2 -1159.272} C_VEL
LIN {X 0,Y 594.473,Z 504.232,A -85,B 0,C 180,E1 -1159.96,E2 -1159.96} C_VEL
LIN {X 0,Y 594.413,Z 514.622,A -85,B 0,C 180,E1 -1160.732,E2 -1160.732} C_VEL
LIN {X 0,Y 594.382,Z 523.132,A -85,B 0,C 180,E1 -1161.502,E2 -1161.502} C_VEL
LIN {X 0,Y 594.346,Z 530.976,A -85,B 0,C 180,E1 -1162.357,E2 -1162.357} C_VEL
LIN {X 0,Y 594.281,Z 538.82,A -85,B 0,C 180,E1 -1163.409,E2 -1163.409} C_VEL
LIN {X 0,Y 594.289,Z 545.689,A -85,B 0,C 180,E1 -1164.573,E2 -1164.573} C_VEL
LIN {X 0,Y 594.27,Z 550.378,A -85,B 0,C 180,E1 -1165.593,E2 -1165.593} C_VEL
LIN {X 0,Y 594.267,Z 553.961,A -85,B 0,C 180,E1 -1166.611,E2 -1166.611} C_VEL
LIN {X 0,Y 594.226,Z 555.812,A -85,B 0,C 180,E1 -1167.29,E2 -1167.29} C_VEL
LIN {X 0,Y 594.241,Z 557.203,A -85,B 0,C 180,E1 -1167.968,E2 -1167.968} C_VEL
LIN {X 0,Y 594.239,Z 558.785,A -85,B 0,C 180,E1 -1169.324,E2 -1169.324} C_VEL
LIN {X 0,Y 594.236,Z 559,A -85,B 0,C 180,E1 -1170.001,E2 -1170.001} C_VEL
LIN {X 0,Y 594.247,Z 558.184,A -85,B 0,C 180,E1 -1171.356,E2 -1171.356} C_VEL
LIN {X 0,Y 594.241,Z 557.2,A -85,B 0,C 180,E1 -1172.034,E2 -1172.034} C_VEL
LIN {X 0,Y 594.226,Z 555.807,A -85,B 0,C 180,E1 -1172.712,E2 -1172.712} C_VEL
LIN {X 0,Y 594.289,Z 552.894,A -85,B 0,C 180,E1 -1173.73,E2 -1173.73} C_VEL
LIN {X 0,Y 594.241,Z 548.947,A -85,B 0,C 180,E1 -1174.749,E2 -1174.749} C_VEL
LIN {X 0,Y 594.304,Z 542.875,A -85,B 0,C 180,E1 -1175.94,E2 -1175.94} C_VEL
LIN {X 0,Y 594.308,Z 536.233,A -85,B 0,C 180,E1 -1176.962,E2 -1176.962} C_VEL
LIN {X 0,Y 594.359,Z 527.987,A -85,B 0,C 180,E1 -1177.987,E2 -1177.987} C_VEL
LIN {X 0,Y 594.382,Z 519.535,A -85,B 0,C 180,E1 -1178.842,E2 -1178.842} C_VEL
LIN {X 0,Y 594.427,Z 509.093,A -85,B 0,C 180,E1 -1179.7,E2 -1179.7} C_VEL
LIN {X 0,Y 594.493,Z 498.758,A -85,B 0,C 180,E1 -1180.386,E2 -1180.386} C_VEL
LIN {X 0,Y 594.559,Z 487.715,A -85,B 0,C 180,E1 -1180.973,E2 -1180.973} C_VEL
LIN {X 0,Y 594.57,Z 475.71,A -85,B 0,C 180,E1 -1181.464,E2 -1181.464} C_VEL
LIN {X 0,Y 594.6,Z 462.355,A -85,B 0,C 180,E1 -1181.851,E2 -1181.851} C_VEL
LIN {X 0,Y 594.676,Z 449.094,A -85,B 0,C 180,E1 -1182.087,E2 -1182.087} C_VEL
LIN {X 0,Y 594.622,Z 347.834,A -85,B 0,C 180,E1 -1183.317,E2 -1183.317} C_VEL
LIN {X 0,Y 594.429,Z 346.271,A -85,B 0,C 180,E1 -1183.351,E2 -1183.351} C_VEL
LIN {X 0,Y 594.526,Z 324.608,A -85,B 0,C 180,E1 -1186.128,E2 -1186.128} C_VEL
LIN {X 0,Y 594.596,Z 302.619,A -85,B 0,C 180,E1 -1188.988,E2 -1188.988} C_VEL
LIN {X 0,Y 594.729,Z 283.67,A -85,B 0,C 180,E1 -1191.488,E2 -1191.488} C_VEL
LIN {X 0,Y 594.777,Z 268.659,A -85,B 0,C 180,E1 -1193.502,E2 -1193.502} C_VEL
LIN {X 0,Y 594.39,Z 266.446,A -85,B 0,C 180,E1 -1193.841,E2 -1193.841} C_VEL
LIN {X 0,Y 594.348,Z 266.454,A -85,B 0,C 180,E1 -1196.7,E2 -1196.7} C_VEL
LIN {X 0,Y 594.368,Z 266.446,A -85,B 0,C 180,E1 -1198.997,E2 -1198.997} C_VEL
LIN {X 0,Y 594.361,Z 266.443,A -85,B 0,C 180,E1 -1201.64,E2 -1201.64} C_VEL
LIN {X 0,Y 594.356,Z 266.446,A -85,B 0,C 180,E1 -1204.134,E2 -1204.134} C_VEL
LIN {X 0,Y 594.339,Z 266.448,A -85,B 0,C 180,E1 -1207.087,E2 -1207.087} C_VEL
LIN {X 0,Y 594.327,Z 266.447,A -85,B 0,C 180,E1 -1209.768,E2 -1209.768} C_VEL
LIN {X 0,Y 594.348,Z 266.45,A -85,B 0,C 180,E1 -1212.373,E2 -1212.373} C_VEL
LIN {X 0,Y 594.316,Z 266.451,A -85,B 0,C 180,E1 -1215.192,E2 -1215.192} C_VEL
LIN {X 0,Y 594.313,Z 266.449,A -85,B 0,C 180,E1 -1217.619,E2 -1217.619} C_VEL
LIN {X 0,Y 594.338,Z 266.45,A -85,B 0,C 180,E1 -1220.316,E2 -1220.316} C_VEL
LIN {X 0,Y 594.352,Z 266.45,A -85,B 0,C 180,E1 -1222.911,E2 -1222.911} C_VEL
LIN {X 0,Y 594.33,Z 266.447,A -85,B 0,C 180,E1 -1225.862,E2 -1225.862} C_VEL
LIN {X 0,Y 594.354,Z 266.454,A -85,B 0,C 180,E1 -1228.648,E2 -1228.648} C_VEL
LIN {X 0,Y 594.339,Z 266.45,A -85,B 0,C 180,E1 -1231.042,E2 -1231.042} C_VEL
LIN {X 0,Y 594.344,Z 266.447,A -85,B 0,C 180,E1 -1233.298,E2 -1233.298} C_VEL
LIN {X 0,Y 594.306,Z 266.45,A -85,B 0,C 180,E1 -1235.574,E2 -1235.574} C_VEL
LIN {X 0,Y 594.322,Z 266.454,A -85,B 0,C 180,E1 -1238.495,E2 -1238.495} C_VEL
LIN {X 0,Y 594.328,Z 266.448,A -85,B 0,C 180,E1 -1241.38,E2 -1241.38} C_VEL
LIN {X 0,Y 594.351,Z 266.444,A -85,B 0,C 180,E1 -1243.513,E2 -1243.513} C_VEL
LIN {X 0,Y 594.341,Z 266.449,A -85,B 0,C 180,E1 -1246.32,E2 -1246.32} C_VEL
LIN {X 0,Y 594.363,Z 266.448,A -85,B 0,C 180,E1 -1249.094,E2 -1249.094} C_VEL
LIN {X 0,Y 594.337,Z 266.446,A -85,B 0,C 180,E1 -1251.842,E2 -1251.842} C_VEL
LIN {X 0,Y 594.372,Z 266.448,A -85,B 0,C 180,E1 -1254.572,E2 -1254.572} C_VEL
LIN {X 0,Y 594.371,Z 266.444,A -85,B 0,C 180,E1 -1257.289,E2 -1257.289} C_VEL
LIN {X 0,Y 594.356,Z 266.444,A -85,B 0,C 180,E1 -1260,E2 -1260} C_VEL
LIN {X 0,Y 594.385,Z 266.449,A -85,B 0,C 180,E1 -1262.711,E2 -1262.711} C_VEL
LIN {X 0,Y 594.364,Z 266.444,A -85,B 0,C 180,E1 -1265.428,E2 -1265.428} C_VEL
LIN {X 0,Y 594.372,Z 266.443,A -85,B 0,C 180,E1 -1268.157,E2 -1268.157} C_VEL
LIN {X 0,Y 594.419,Z 266.441,A -85,B 0,C 180,E1 -1271.112,E2 -1271.112} C_VEL
LIN {X 0,Y 594.345,Z 266.446,A -85,B 0,C 180,E1 -1274.175,E2 -1274.175} C_VEL
LIN {X 0,Y 594.335,Z 266.449,A -85,B 0,C 180,E1 -1275.353,E2 -1275.353} C_VEL
LIN {X 0,Y 593.663,Z 266.532,A -85,B 0,C 180,E1 -1275.919,E2 -1275.919} C_VEL
LIN {X 0,Y 590.804,Z 266.896,A -85,B 0,C 180,E1 -1276.837,E2 -1276.837} C_VEL
LIN {X 0,Y 588.398,Z 267.19,A -85,B 0,C 180,E1 -1277.576,E2 -1277.576} C_VEL
LIN {X 0,Y 587.375,Z 267.314,A -85,B 0,C 180,E1 -1278.146,E2 -1278.146} C_VEL
LIN {X 0,Y 587.297,Z 267.325,A -85,B 0,C 180,E1 -1278.339,E2 -1278.339} C_VEL
LIN {X 0,Y 587.318,Z 267.328,A -85,B 0,C 180,E1 -1281.046,E2 -1281.046} C_VEL
LIN {X 0,Y 587.301,Z 267.323,A -85,B 0,C 180,E1 -1284.008,E2 -1284.008} C_VEL
LIN {X 0,Y 587.33,Z 267.321,A -85,B 0,C 180,E1 -1286.279,E2 -1286.279} C_VEL
LIN {X 0,Y 587.323,Z 267.326,A -85,B 0,C 180,E1 -1289.137,E2 -1289.137} C_VEL
LIN {X 0,Y 587.325,Z 267.319,A -85,B 0,C 180,E1 -1291.84,E2 -1291.84} C_VEL
LIN {X 0,Y 587.331,Z 267.321,A -85,B 0,C 180,E1 -1294.352,E2 -1294.352} C_VEL
LIN {X 0,Y 587.327,Z 267.327,A -85,B 0,C 180,E1 -1296.748,E2 -1296.748} C_VEL
LIN {X 0,Y 587.324,Z 267.323,A -85,B 0,C 180,E1 -1299.361,E2 -1299.361} C_VEL
LIN {X 0,Y 587.309,Z 267.322,A -85,B 0,C 180,E1 -1302.11,E2 -1302.11} C_VEL
LIN {X 0,Y 587.293,Z 267.332,A -85,B 0,C 180,E1 -1305.091,E2 -1305.091} C_VEL
LIN {X 0,Y 587.332,Z 267.319,A -85,B 0,C 180,E1 -1307.929,E2 -1307.929} C_VEL
LIN {X 0,Y 587.33,Z 267.324,A -85,B 0,C 180,E1 -1310.643,E2 -1310.643} C_VEL
LIN {X 0,Y 587.34,Z 267.323,A -85,B 0,C 180,E1 -1313.293,E2 -1313.293} C_VEL
LIN {X 0,Y 587.329,Z 267.319,A -85,B 0,C 180,E1 -1315.78,E2 -1315.78} C_VEL
LIN {X 0,Y 587.337,Z 267.319,A -85,B 0,C 180,E1 -1318.233,E2 -1318.233} C_VEL
LIN {X 0,Y 587.341,Z 267.326,A -85,B 0,C 180,E1 -1320.867,E2 -1320.867} C_VEL
LIN {X 0,Y 587.349,Z 267.317,A -85,B 0,C 180,E1 -1323.82,E2 -1323.82} C_VEL
LIN {X 0,Y 587.329,Z 267.319,A -85,B 0,C 180,E1 -1325.995,E2 -1325.995} C_VEL
LIN {X 0,Y 587.314,Z 267.321,A -85,B 0,C 180,E1 -1328.227,E2 -1328.227} C_VEL
LIN {X 0,Y 587.346,Z 267.325,A -85,B 0,C 180,E1 -1331.152,E2 -1331.152} C_VEL
LIN {X 0,Y 587.32,Z 267.32,A -85,B 0,C 180,E1 -1334.025,E2 -1334.025} C_VEL
LIN {X 0,Y 587.354,Z 267.316,A -85,B 0,C 180,E1 -1336.154,E2 -1336.154} C_VEL
LIN {X 0,Y 587.341,Z 267.326,A -85,B 0,C 180,E1 -1338.962,E2 -1338.962} C_VEL
LIN {X 0,Y 587.367,Z 267.315,A -85,B 0,C 180,E1 -1341.744,E2 -1341.744} C_VEL
LIN {X 0,Y 587.352,Z 267.318,A -85,B 0,C 180,E1 -1344.506,E2 -1344.506} C_VEL
LIN {X 0,Y 587.37,Z 267.321,A -85,B 0,C 180,E1 -1347.256,E2 -1347.256} C_VEL
LIN {X 0,Y 587.382,Z 267.312,A -85,B 0,C 180,E1 -1349.999,E2 -1349.999} C_VEL
LIN {X 0,Y 587.367,Z 267.319,A -85,B 0,C 180,E1 -1352.742,E2 -1352.742} C_VEL
LIN {X 0,Y 587.362,Z 267.319,A -85,B 0,C 180,E1 -1355.491,E2 -1355.491} C_VEL
LIN {X 0,Y 587.361,Z 267.315,A -85,B 0,C 180,E1 -1358.253,E2 -1358.253} C_VEL
LIN {X 0,Y 587.341,Z 267.328,A -85,B 0,C 180,E1 -1361.132,E2 -1361.132} C_VEL
LIN {X 0,Y 587.357,Z 267.315,A -85,B 0,C 180,E1 -1364.258,E2 -1364.258} C_VEL
LIN {X 0,Y 587.35,Z 267.322,A -85,B 0,C 180,E1 -1367.403,E2 -1367.403} C_VEL
LIN {X 0,Y 587.324,Z 267.319,A -85,B 0,C 180,E1 -1370.302,E2 -1370.302} C_VEL
LIN {X 0,Y 587.354,Z 267.325,A -85,B 0,C 180,E1 -1373.254,E2 -1373.254} C_VEL
LIN {X 0,Y 587.348,Z 267.316,A -85,B 0,C 180,E1 -1376.274,E2 -1376.274} C_VEL
LIN {X 0,Y 587.338,Z 267.327,A -85,B 0,C 180,E1 -1379.132,E2 -1379.132} C_VEL
LIN {X 0,Y 587.342,Z 267.318,A -85,B 0,C 180,E1 -1381.836,E2 -1381.836} C_VEL
LIN {X 0,Y 587.338,Z 267.318,A -85,B 0,C 180,E1 -1384.347,E2 -1384.347} C_VEL
LIN {X 0,Y 587.328,Z 267.322,A -85,B 0,C 180,E1 -1386.743,E2 -1386.743} C_VEL
LIN {X 0,Y 587.325,Z 267.328,A -85,B 0,C 180,E1 -1389.355,E2 -1389.355} C_VEL
LIN {X 0,Y 587.331,Z 267.319,A -85,B 0,C 180,E1 -1392.108,E2 -1392.108} C_VEL
LIN {X 0,Y 587.375,Z 267.445,A -85,B 0,C 180,E1 -1394.527,E2 -1394.527} C_VEL
LIN {X 0,Y 587.329,Z 281.734,A -85,B 0,C 180,E1 -1397.23,E2 -1397.23} C_VEL
LIN {X 0,Y 587.299,Z 288.907,A -85,B 0,C 180,E1 -1398.572,E2 -1398.572} C_VEL
LIN {X 0,Y 587.839,Z 292.773,A -85,B 0,C 180,E1 -1398.633,E2 -1398.633} C_VEL
LIN {X 0,Y 587.716,Z 395.067,A -85,B 0,C 180,E1 -1399.902,E2 -1399.902} C_VEL
LIN {X 0,Y 587.665,Z 408.826,A -85,B 0,C 180,E1 -1400.222,E2 -1400.222} C_VEL
LIN {X 0,Y 587.606,Z 421.45,A -85,B 0,C 180,E1 -1400.662,E2 -1400.662} C_VEL
LIN {X 0,Y 587.536,Z 432.175,A -85,B 0,C 180,E1 -1401.163,E2 -1401.163} C_VEL
LIN {X 0,Y 587.445,Z 442.721,A -85,B 0,C 180,E1 -1401.784,E2 -1401.784} C_VEL
LIN {X 0,Y 587.404,Z 452.642,A -85,B 0,C 180,E1 -1402.505,E2 -1402.505} C_VEL
LIN {X 0,Y 587.337,Z 462.051,A -85,B 0,C 180,E1 -1403.34,E2 -1403.34} C_VEL
LIN {X 0,Y 587.279,Z 470.959,A -85,B 0,C 180,E1 -1404.308,E2 -1404.308} C_VEL
LIN {X 0,Y 587.238,Z 478.508,A -85,B 0,C 180,E1 -1405.328,E2 -1405.328} C_VEL
LIN {X 0,Y 587.208,Z 484.823,A -85,B 0,C 180,E1 -1406.39,E2 -1406.39} C_VEL
LIN {X 0,Y 587.154,Z 489.636,A -85,B 0,C 180,E1 -1407.41,E2 -1407.41} C_VEL
LIN {X 0,Y 587.176,Z 493.971,A -85,B 0,C 180,E1 -1408.624,E2 -1408.624} C_VEL
LIN {X 0,Y 587.158,Z 496.899,A -85,B 0,C 180,E1 -1409.82,E2 -1409.82} C_VEL
LIN {X 0,Y 587.155,Z 498.425,A -85,B 0,C 180,E1 -1410.888,E2 -1410.888} C_VEL
LIN {X 0,Y 587.126,Z 498.94,A -85,B 0,C 180,E1 -1412.336,E2 -1412.336} C_VEL
LIN {X 0,Y 587.127,Z 498.641,A -85,B 0,C 180,E1 -1412.944,E2 -1412.944} C_VEL
LIN {X 0,Y 587.137,Z 497.612,A -85,B 0,C 180,E1 -1413.849,E2 -1413.849} C_VEL
LIN {X 0,Y 587.156,Z 494.672,A -85,B 0,C 180,E1 -1415.233,E2 -1415.233} C_VEL
LIN {X 0,Y 587.181,Z 490.943,A -85,B 0,C 180,E1 -1416.362,E2 -1416.362} C_VEL
LIN {X 0,Y 587.187,Z 485.963,A -85,B 0,C 180,E1 -1417.48,E2 -1417.48} C_VEL
LIN {X 0,Y 587.235,Z 479.617,A -85,B 0,C 180,E1 -1418.591,E2 -1418.591} C_VEL
LIN {X 0,Y 587.265,Z 471.674,A -85,B 0,C 180,E1 -1419.693,E2 -1419.693} C_VEL
LIN {X 0,Y 587.326,Z 462.284,A -85,B 0,C 180,E1 -1420.728,E2 -1420.728} C_VEL
LIN {X 0,Y 587.408,Z 452.378,A -85,B 0,C 180,E1 -1421.606,E2 -1421.606} C_VEL
LIN {X 0,Y 587.421,Z 442.407,A -85,B 0,C 180,E1 -1422.327,E2 -1422.327} C_VEL
LIN {X 0,Y 587.557,Z 430.699,A -85,B 0,C 180,E1 -1423.003,E2 -1423.003} C_VEL
LIN {X 0,Y 587.597,Z 417.34,A -85,B 0,C 180,E1 -1423.587,E2 -1423.587} C_VEL
LIN {X 0,Y 587.651,Z 405.148,A -85,B 0,C 180,E1 -1423.967,E2 -1423.967} C_VEL
LIN {X 0,Y 587.708,Z 393.491,A -85,B 0,C 180,E1 -1424.214,E2 -1424.214} C_VEL
LIN {X 0,Y 587.704,Z 291.304,A -85,B 0,C 180,E1 -1425.479,E2 -1425.479} C_VEL
LIN {X 0,Y 587.327,Z 288.798,A -85,B 0,C 180,E1 -1425.536,E2 -1425.536} C_VEL
LIN {X 0,Y 587.349,Z 274.293,A -85,B 0,C 180,E1 -1428.264,E2 -1428.264} C_VEL
LIN {X 0,Y 587.296,Z 267.326,A -85,B 0,C 180,E1 -1429.616,E2 -1429.616} C_VEL
LIN {X 0,Y 587.325,Z 267.323,A -85,B 0,C 180,E1 -1432.437,E2 -1432.437} C_VEL
LIN {X 0,Y 587.316,Z 267.327,A -85,B 0,C 180,E1 -1435.195,E2 -1435.195} C_VEL
LIN {X 0,Y 587.295,Z 267.323,A -85,B 0,C 180,E1 -1437.943,E2 -1437.943} C_VEL
LIN {X 0,Y 587.351,Z 267.322,A -85,B 0,C 180,E1 -1440.686,E2 -1440.686} C_VEL
LIN {X 0,Y 587.296,Z 267.326,A -85,B 0,C 180,E1 -1443.431,E2 -1443.431} C_VEL
LIN {X 0,Y 587.316,Z 267.323,A -85,B 0,C 180,E1 -1445.494,E2 -1445.494} C_VEL
LIN {X 0,Y 587.31,Z 267.322,A -85,B 0,C 180,E1 -1448.256,E2 -1448.256} C_VEL
LIN {X 0,Y 587.366,Z 267.322,A -85,B 0,C 180,E1 -1451.177,E2 -1451.177} C_VEL
LIN {X 0,Y 587.303,Z 267.322,A -85,B 0,C 180,E1 -1454.263,E2 -1454.263} C_VEL
LIN {X 0,Y 587.309,Z 267.325,A -85,B 0,C 180,E1 -1457.408,E2 -1457.408} C_VEL
LIN {X 0,Y 587.296,Z 267.325,A -85,B 0,C 180,E1 -1459.577,E2 -1459.577} C_VEL
LIN {X 0,Y 587.281,Z 267.325,A -85,B 0,C 180,E1 -1461.776,E2 -1461.776} C_VEL
LIN {X 0,Y 587.301,Z 267.327,A -85,B 0,C 180,E1 -1464.761,E2 -1464.761} C_VEL
LIN {X 0,Y 587.299,Z 267.331,A -85,B 0,C 180,E1 -1467.048,E2 -1467.048} C_VEL
LIN {X 0,Y 587.3,Z 267.329,A -85,B 0,C 180,E1 -1469.382,E2 -1469.382} C_VEL
LIN {X 0,Y 587.308,Z 267.322,A -85,B 0,C 180,E1 -1471.841,E2 -1471.841} C_VEL
LIN {X 0,Y 587.311,Z 267.321,A -85,B 0,C 180,E1 -1474.353,E2 -1474.353} C_VEL
LIN {X 0,Y 587.309,Z 267.324,A -85,B 0,C 180,E1 -1476.75,E2 -1476.75} C_VEL
LIN {X 0,Y 587.31,Z 267.329,A -85,B 0,C 180,E1 -1479.363,E2 -1479.363} C_VEL
LIN {X 0,Y 587.297,Z 267.322,A -85,B 0,C 180,E1 -1482.112,E2 -1482.112} C_VEL
LIN {X 0,Y 587.282,Z 267.332,A -85,B 0,C 180,E1 -1485.093,E2 -1485.093} C_VEL
LIN {X 0,Y 587.322,Z 267.321,A -85,B 0,C 180,E1 -1487.931,E2 -1487.931} C_VEL
LIN {X 0,Y 587.294,Z 267.329,A -85,B 0,C 180,E1 -1491.064,E2 -1491.064} C_VEL
LIN {X 0,Y 587.323,Z 267.33,A -85,B 0,C 180,E1 -1493.296,E2 -1493.296} C_VEL
LIN {X 0,Y 587.338,Z 267.322,A -85,B 0,C 180,E1 -1495.784,E2 -1495.784} C_VEL
LIN {X 0,Y 587.323,Z 267.321,A -85,B 0,C 180,E1 -1498.235,E2 -1498.235} C_VEL
LIN {X 0,Y 587.333,Z 267.322,A -85,B 0,C 180,E1 -1500.87,E2 -1500.87} C_VEL
LIN {X 0,Y 587.32,Z 267.325,A -85,B 0,C 180,E1 -1503.828,E2 -1503.828} C_VEL
LIN {X 0,Y 587.385,Z 267.483,A -85,B 0,C 180,E1 -1506.023,E2 -1506.023} C_VEL
LIN {X 0,Y 587.955,Z 271.406,A -85,B 0,C 180,E1 -1506.585,E2 -1506.585} C_VEL
LIN {X 0,Y 587.786,Z 293.24,A -85,B 0,C 180,E1 -1509.532,E2 -1509.532} C_VEL
LIN {X 0,Y 587.585,Z 315.073,A -85,B 0,C 180,E1 -1512.425,E2 -1512.425} C_VEL
LIN {X 0,Y 587.484,Z 334.178,A -85,B 0,C 180,E1 -1514.921,E2 -1514.921} C_VEL
LIN {X 0,Y 587.386,Z 346.452,A -85,B 0,C 180,E1 -1516.499,E2 -1516.499} C_VEL
LIN {X 0,Y 587.833,Z 350.923,A -85,B 0,C 180,E1 -1516.565,E2 -1516.565} C_VEL
LIN {X 0,Y 587.722,Z 455.07,A -85,B 0,C 180,E1 -1517.857,E2 -1517.857} C_VEL
LIN {X 0,Y 587.669,Z 468.3,A -85,B 0,C 180,E1 -1518.163,E2 -1518.163} C_VEL
LIN {X 0,Y 587.614,Z 480.994,A -85,B 0,C 180,E1 -1518.599,E2 -1518.599} C_VEL
LIN {X 0,Y 587.548,Z 492.671,A -85,B 0,C 180,E1 -1519.143,E2 -1519.143} C_VEL
LIN {X 0,Y 587.469,Z 504.233,A -85,B 0,C 180,E1 -1519.839,E2 -1519.839} C_VEL
LIN {X 0,Y 587.392,Z 514.623,A -85,B 0,C 180,E1 -1520.62,E2 -1520.62} C_VEL
LIN {X 0,Y 587.321,Z 523.133,A -85,B 0,C 180,E1 -1521.4,E2 -1521.4} C_VEL
LIN {X 0,Y 587.273,Z 530.976,A -85,B 0,C 180,E1 -1522.265,E2 -1522.265} C_VEL
LIN {X 0,Y 587.231,Z 537.482,A -85,B 0,C 180,E1 -1523.128,E2 -1523.128} C_VEL
LIN {X 0,Y 587.236,Z 543.876,A -85,B 0,C 180,E1 -1524.163,E2 -1524.163} C_VEL
LIN {X 0,Y 587.147,Z 548.956,A -85,B 0,C 180,E1 -1525.195,E2 -1525.195} C_VEL
LIN {X 0,Y 587.213,Z 552.9,A -85,B 0,C 180,E1 -1526.227,E2 -1526.227} C_VEL
LIN {X 0,Y 587.132,Z 555.812,A -85,B 0,C 180,E1 -1527.257,E2 -1527.257} C_VEL
LIN {X 0,Y 587.14,Z 557.202,A -85,B 0,C 180,E1 -1527.943,E2 -1527.943} C_VEL
LIN {X 0,Y 587.14,Z 558.785,A -85,B 0,C 180,E1 -1529.315,E2 -1529.315} C_VEL
LIN {X 0,Y 587.137,Z 559,A -85,B 0,C 180,E1 -1530.001,E2 -1530.001} C_VEL
LIN {X 0,Y 587.147,Z 558.184,A -85,B 0,C 180,E1 -1531.373,E2 -1531.373} C_VEL
LIN {X 0,Y 587.14,Z 557.199,A -85,B 0,C 180,E1 -1532.059,E2 -1532.059} C_VEL
LIN {X 0,Y 587.132,Z 555.808,A -85,B 0,C 180,E1 -1532.745,E2 -1532.745} C_VEL
LIN {X 0,Y 587.213,Z 552.894,A -85,B 0,C 180,E1 -1533.775,E2 -1533.775} C_VEL
LIN {X 0,Y 587.147,Z 548.947,A -85,B 0,C 180,E1 -1534.807,E2 -1534.807} C_VEL
LIN {X 0,Y 587.217,Z 542.874,A -85,B 0,C 180,E1 -1536.012,E2 -1536.012} C_VEL
LIN {X 0,Y 587.245,Z 536.234,A -85,B 0,C 180,E1 -1537.047,E2 -1537.047} C_VEL
LIN {X 0,Y 587.3,Z 527.988,A -85,B 0,C 180,E1 -1538.083,E2 -1538.083} C_VEL
LIN {X 0,Y 587.343,Z 519.536,A -85,B 0,C 180,E1 -1538.949,E2 -1538.949} C_VEL
LIN {X 0,Y 587.414,Z 509.094,A -85,B 0,C 180,E1 -1539.816,E2 -1539.816} C_VEL
LIN {X 0,Y 587.51,Z 498.757,A -85,B 0,C 180,E1 -1540.511,E2 -1540.511} C_VEL
LIN {X 0,Y 587.568,Z 486.983,A -85,B 0,C 180,E1 -1541.141,E2 -1541.141} C_VEL
LIN {X 0,Y 587.604,Z 474.601,A -85,B 0,C 180,E1 -1541.64,E2 -1541.64} C_VEL
LIN {X 0,Y 587.683,Z 461.44,A -85,B 0,C 180,E1 -1542.014,E2 -1542.014} C_VEL
LIN {X 0,Y 587.758,Z 449.094,A -85,B 0,C 180,E1 -1542.232,E2 -1542.232} C_VEL
LIN {X 0,Y 587.714,Z 348.504,A -85,B 0,C 180,E1 -1543.468,E2 -1543.468} C_VEL
LIN {X 0,Y 587.394,Z 346.271,A -85,B 0,C 180,E1 -1543.514,E2 -1543.514} C_VEL
LIN {X 0,Y 587.551,Z 325.973,A -85,B 0,C 180,E1 -1546.147,E2 -1546.147} C_VEL
LIN {X 0,Y 587.643,Z 305.504,A -85,B 0,C 180,E1 -1548.838,E2 -1548.838} C_VEL
LIN {X 0,Y 587.859,Z 286.323,A -85,B 0,C 180,E1 -1551.394,E2 -1551.394} C_VEL
LIN {X 0,Y 587.965,Z 271.388,A -85,B 0,C 180,E1 -1553.417,E2 -1553.417} C_VEL
LIN {X 0,Y 587.346,Z 267.324,A -85,B 0,C 180,E1 -1554.005,E2 -1554.005} C_VEL
LIN {X 0,Y 587.291,Z 267.327,A -85,B 0,C 180,E1 -1557.046,E2 -1557.046} C_VEL
LIN {X 0,Y 587.305,Z 267.322,A -85,B 0,C 180,E1 -1559.38,E2 -1559.38} C_VEL
LIN {X 0,Y 587.332,Z 267.319,A -85,B 0,C 180,E1 -1561.833,E2 -1561.833} C_VEL
LIN {X 0,Y 587.326,Z 267.325,A -85,B 0,C 180,E1 -1564.344,E2 -1564.344} C_VEL
LIN {X 0,Y 587.296,Z 267.323,A -85,B 0,C 180,E1 -1567.608,E2 -1567.608} C_VEL
LIN {X 0,Y 587.289,Z 267.328,A -85,B 0,C 180,E1 -1570.253,E2 -1570.253} C_VEL
LIN {X 0,Y 587.286,Z 267.328,A -85,B 0,C 180,E1 -1573.005,E2 -1573.005} C_VEL
LIN {X 0,Y 587.291,Z 267.325,A -85,B 0,C 180,E1 -1576.046,E2 -1576.046} C_VEL
LIN {X 0,Y 587.313,Z 267.327,A -85,B 0,C 180,E1 -1578.923,E2 -1578.923} C_VEL
LIN {X 0,Y 587.287,Z 267.324,A -85,B 0,C 180,E1 -1581.517,E2 -1581.517} C_VEL
LIN {X 0,Y 587.257,Z 267.33,A -85,B 0,C 180,E1 -1584.097,E2 -1584.097} C_VEL
LIN {X 0,Y 587.305,Z 267.329,A -85,B 0,C 180,E1 -1586.887,E2 -1586.887} C_VEL
LIN {X 0,Y 587.291,Z 267.324,A -85,B 0,C 180,E1 -1589.49,E2 -1589.49} C_VEL
LIN {X 0,Y 587.315,Z 267.324,A -85,B 0,C 180,E1 -1592.305,E2 -1592.305} C_VEL
LIN {X 0,Y 587.266,Z 267.329,A -85,B 0,C 180,E1 -1595.237,E2 -1595.237} C_VEL
LIN {X 0,Y 587.271,Z 267.327,A -85,B 0,C 180,E1 -1597.483,E2 -1597.483} C_VEL
LIN {X 0,Y 587.279,Z 267.325,A -85,B 0,C 180,E1 -1599.693,E2 -1599.693} C_VEL
LIN {X 0,Y 587.311,Z 267.329,A -85,B 0,C 180,E1 -1602.593,E2 -1602.593} C_VEL
LIN {X 0,Y 587.296,Z 267.324,A -85,B 0,C 180,E1 -1605.445,E2 -1605.445} C_VEL
LIN {X 0,Y 587.302,Z 267.325,A -85,B 0,C 180,E1 -1608.262,E2 -1608.262} C_VEL
LIN {X 0,Y 587.309,Z 267.327,A -85,B 0,C 180,E1 -1611.05,E2 -1611.05} C_VEL
LIN {X 0,Y 587.329,Z 267.322,A -85,B 0,C 180,E1 -1613.265,E2 -1613.265} C_VEL
LIN {X 0,Y 587.26,Z 267.328,A -85,B 0,C 180,E1 -1615.882,E2 -1615.882} C_VEL
LIN {X 0,Y 587.311,Z 267.321,A -85,B 0,C 180,E1 -1617.942,E2 -1617.942} C_VEL
LIN {X 0,Y 587.371,Z 267.322,A -85,B 0,C 180,E1 -1620.685,E2 -1620.685} C_VEL
LIN {X 0,Y 587.303,Z 267.324,A -85,B 0,C 180,E1 -1623.43,E2 -1623.43} C_VEL
LIN {X 0,Y 587.326,Z 267.32,A -85,B 0,C 180,E1 -1625.493,E2 -1625.493} C_VEL
LIN {X 0,Y 587.328,Z 267.321,A -85,B 0,C 180,E1 -1628.255,E2 -1628.255} C_VEL
LIN {X 0,Y 587.387,Z 267.317,A -85,B 0,C 180,E1 -1631.176,E2 -1631.176} C_VEL
LIN {X 0,Y 587.322,Z 267.322,A -85,B 0,C 180,E1 -1634.262,E2 -1634.262} C_VEL
LIN {X 0,Y 587.325,Z 267.322,A -85,B 0,C 180,E1 -1637.406,E2 -1637.406} C_VEL
LIN {X 0,Y 587.297,Z 267.325,A -85,B 0,C 180,E1 -1638.339,E2 -1638.339} C_VEL
LIN {X 0,Y 586.649,Z 267.414,A -85,B 0,C 180,E1 -1638.911,E2 -1638.911} C_VEL
LIN {X 0,Y 583.814,Z 267.768,A -85,B 0,C 180,E1 -1639.839,E2 -1639.839} C_VEL
LIN {X 0,Y 581.398,Z 268.067,A -85,B 0,C 180,E1 -1640.586,E2 -1640.586} C_VEL
LIN {X 0,Y 580.345,Z 268.195,A -85,B 0,C 180,E1 -1641.163,E2 -1641.163} C_VEL
LIN {X 0,Y 580.251,Z 268.204,A -85,B 0,C 180,E1 -1641.358,E2 -1641.358} C_VEL
LIN {X 0,Y 580.264,Z 268.201,A -85,B 0,C 180,E1 -1644.317,E2 -1644.317} C_VEL
LIN {X 0,Y 580.279,Z 268.203,A -85,B 0,C 180,E1 -1646.623,E2 -1646.623} C_VEL
LIN {X 0,Y 580.276,Z 268.201,A -85,B 0,C 180,E1 -1649.313,E2 -1649.313} C_VEL
LIN {X 0,Y 580.272,Z 268.199,A -85,B 0,C 180,E1 -1652.202,E2 -1652.202} C_VEL
LIN {X 0,Y 580.275,Z 268.205,A -85,B 0,C 180,E1 -1654.697,E2 -1654.697} C_VEL
LIN {X 0,Y 580.274,Z 268.203,A -85,B 0,C 180,E1 -1657.27,E2 -1657.27} C_VEL
LIN {X 0,Y 580.274,Z 268.199,A -85,B 0,C 180,E1 -1660.274,E2 -1660.274} C_VEL
LIN {X 0,Y 580.259,Z 268.206,A -85,B 0,C 180,E1 -1662.707,E2 -1662.707} C_VEL
LIN {X 0,Y 580.251,Z 268.202,A -85,B 0,C 180,E1 -1665.61,E2 -1665.61} C_VEL
LIN {X 0,Y 580.301,Z 268.195,A -85,B 0,C 180,E1 -1668.237,E2 -1668.237} C_VEL
LIN {X 0,Y 580.276,Z 268.207,A -85,B 0,C 180,E1 -1670.968,E2 -1670.968} C_VEL
LIN {X 0,Y 580.282,Z 268.198,A -85,B 0,C 180,E1 -1673.6,E2 -1673.6} C_VEL
LIN {X 0,Y 580.291,Z 268.196,A -85,B 0,C 180,E1 -1676.146,E2 -1676.146} C_VEL
LIN {X 0,Y 580.272,Z 268.203,A -85,B 0,C 180,E1 -1678.616,E2 -1678.616} C_VEL
LIN {X 0,Y 580.286,Z 268.206,A -85,B 0,C 180,E1 -1681.025,E2 -1681.025} C_VEL
LIN {X 0,Y 580.283,Z 268.198,A -85,B 0,C 180,E1 -1683.667,E2 -1683.667} C_VEL
LIN {X 0,Y 580.293,Z 268.197,A -85,B 0,C 180,E1 -1685.685,E2 -1685.685} C_VEL
LIN {X 0,Y 580.265,Z 268.199,A -85,B 0,C 180,E1 -1687.948,E2 -1687.948} C_VEL
LIN {X 0,Y 580.314,Z 268.202,A -85,B 0,C 180,E1 -1690.915,E2 -1690.915} C_VEL
LIN {X 0,Y 580.275,Z 268.198,A -85,B 0,C 180,E1 -1693.826,E2 -1693.826} C_VEL
LIN {X 0,Y 580.321,Z 268.192,A -85,B 0,C 180,E1 -1695.983,E2 -1695.983} C_VEL
LIN {X 0,Y 580.302,Z 268.201,A -85,B 0,C 180,E1 -1698.827,E2 -1698.827} C_VEL
LIN {X 0,Y 580.33,Z 268.193,A -85,B 0,C 180,E1 -1701.644,E2 -1701.644} C_VEL
LIN {X 0,Y 580.318,Z 268.194,A -85,B 0,C 180,E1 -1704.44,E2 -1704.44} C_VEL
LIN {X 0,Y 580.341,Z 268.19,A -85,B 0,C 180,E1 -1707.917,E2 -1707.917} C_VEL
LIN {X 0,Y 580.356,Z 268.191,A -85,B 0,C 180,E1 -1710.693,E2 -1710.693} C_VEL
LIN {X 0,Y 580.286,Z 268.201,A -85,B 0,C 180,E1 -1713.47,E2 -1713.47} C_VEL
LIN {X 0,Y 580.328,Z 268.194,A -85,B 0,C 180,E1 -1715.558,E2 -1715.558} C_VEL
LIN {X 0,Y 580.324,Z 268.192,A -85,B 0,C 180,E1 -1718.354,E2 -1718.354} C_VEL
LIN {X 0,Y 580.293,Z 268.205,A -85,B 0,C 180,E1 -1721.189,E2 -1721.189} C_VEL
LIN {X 0,Y 580.32,Z 268.192,A -85,B 0,C 180,E1 -1724.014,E2 -1724.014} C_VEL
LIN {X 0,Y 580.304,Z 268.2,A -85,B 0,C 180,E1 -1726.912,E2 -1726.912} C_VEL
LIN {X 0,Y 580.298,Z 268.196,A -85,B 0,C 180,E1 -1729.819,E2 -1729.819} C_VEL
LIN {X 0,Y 580.316,Z 268.197,A -85,B 0,C 180,E1 -1732.798,E2 -1732.798} C_VEL
LIN {X 0,Y 580.294,Z 268.204,A -85,B 0,C 180,E1 -1735.076,E2 -1735.076} C_VEL
LIN {X 0,Y 580.303,Z 268.195,A -85,B 0,C 180,E1 -1737.86,E2 -1737.86} C_VEL
LIN {X 0,Y 580.281,Z 268.199,A -85,B 0,C 180,E1 -1740.695,E2 -1740.695} C_VEL
LIN {X 0,Y 580.287,Z 268.204,A -85,B 0,C 180,E1 -1743.314,E2 -1743.314} C_VEL
LIN {X 0,Y 580.303,Z 268.196,A -85,B 0,C 180,E1 -1745.765,E2 -1745.765} C_VEL
LIN {X 0,Y 580.264,Z 268.199,A -85,B 0,C 180,E1 -1748.142,E2 -1748.142} C_VEL
LIN {X 0,Y 580.292,Z 268.2,A -85,B 0,C 180,E1 -1750.837,E2 -1750.837} C_VEL
LIN {X 0,Y 580.267,Z 268.205,A -85,B 0,C 180,E1 -1753.652,E2 -1753.652} C_VEL
LIN {X 0,Y 580.336,Z 268.31,A -85,B 0,C 180,E1 -1754.474,E2 -1754.474} C_VEL
LIN {X 0,Y 580.266,Z 281.199,A -85,B 0,C 180,E1 -1756.943,E2 -1756.943} C_VEL
LIN {X 0,Y 580.296,Z 288.868,A -85,B 0,C 180,E1 -1758.4,E2 -1758.4} C_VEL
LIN {X 0,Y 580.935,Z 294.876,A -85,B 0,C 180,E1 -1758.496,E2 -1758.496} C_VEL
LIN {X 0,Y 580.792,Z 394.98,A -85,B 0,C 180,E1 -1759.754,E2 -1759.754} C_VEL
LIN {X 0,Y 580.717,Z 408.194,A -85,B 0,C 180,E1 -1760.06,E2 -1760.06} C_VEL
LIN {X 0,Y 580.627,Z 421.317,A -85,B 0,C 180,E1 -1760.518,E2 -1760.518} C_VEL
LIN {X 0,Y 580.513,Z 433.334,A -85,B 0,C 180,E1 -1761.096,E2 -1761.096} C_VEL
LIN {X 0,Y 580.403,Z 444.095,A -85,B 0,C 180,E1 -1761.753,E2 -1761.753} C_VEL
LIN {X 0,Y 580.373,Z 454.231,A -85,B 0,C 180,E1 -1762.519,E2 -1762.519} C_VEL
LIN {X 0,Y 580.273,Z 463.768,A -85,B 0,C 180,E1 -1763.403,E2 -1763.403} C_VEL
LIN {X 0,Y 580.189,Z 472.807,A -85,B 0,C 180,E1 -1764.449,E2 -1764.449} C_VEL
LIN {X 0,Y 580.155,Z 479.815,A -85,B 0,C 180,E1 -1765.452,E2 -1765.452} C_VEL
LIN {X 0,Y 580.129,Z 485.453,A -85,B 0,C 180,E1 -1766.445,E2 -1766.445} C_VEL
LIN {X 0,Y 580.066,Z 489.715,A -85,B 0,C 180,E1 -1767.374,E2 -1767.374} C_VEL
LIN {X 0,Y 580.068,Z 492.11,A -85,B 0,C 180,E1 -1767.995,E2 -1767.995} C_VEL
LIN {X 0,Y 580.067,Z 495.915,A -85,B 0,C 180,E1 -1769.33,E2 -1769.33} C_VEL
LIN {X 0,Y 580.048,Z 497.606,A -85,B 0,C 180,E1 -1770.214,E2 -1770.214} C_VEL
LIN {X 0,Y 580.059,Z 498.559,A -85,B 0,C 180,E1 -1771.012,E2 -1771.012} C_VEL
LIN {X 0,Y 580.02,Z 498.976,A -85,B 0,C 180,E1 -1772.18,E2 -1772.18} C_VEL
LIN {X 0,Y 580.052,Z 497.837,A -85,B 0,C 180,E1 -1773.7,E2 -1773.7} C_VEL
LIN {X 0,Y 580.051,Z 495.59,A -85,B 0,C 180,E1 -1774.909,E2 -1774.909} C_VEL
LIN {X 0,Y 580.11,Z 492.248,A -85,B 0,C 180,E1 -1776.056,E2 -1776.056} C_VEL
LIN {X 0,Y 580.115,Z 487.69,A -85,B 0,C 180,E1 -1777.191,E2 -1777.191} C_VEL
LIN {X 0,Y 580.154,Z 481.8,A -85,B 0,C 180,E1 -1778.317,E2 -1778.317} C_VEL
LIN {X 0,Y 580.22,Z 474.341,A -85,B 0,C 180,E1 -1779.436,E2 -1779.436} C_VEL
LIN {X 0,Y 580.258,Z 466.762,A -85,B 0,C 180,E1 -1780.361,E2 -1780.361} C_VEL
LIN {X 0,Y 580.331,Z 457.577,A -85,B 0,C 180,E1 -1781.282,E2 -1781.282} C_VEL
LIN {X 0,Y 580.382,Z 446.155,A -85,B 0,C 180,E1 -1782.197,E2 -1782.197} C_VEL
LIN {X 0,Y 580.518,Z 435.274,A -85,B 0,C 180,E1 -1782.885,E2 -1782.885} C_VEL
LIN {X 0,Y 580.584,Z 424.548,A -85,B 0,C 180,E1 -1783.428,E2 -1783.428} C_VEL
LIN {X 0,Y 580.64,Z 412.956,A -85,B 0,C 180,E1 -1783.881,E2 -1783.881} C_VEL
LIN {X 0,Y 580.737,Z 399.758,A -85,B 0,C 180,E1 -1784.245,E2 -1784.245} C_VEL
LIN {X 0,Y 580.803,Z 385.396,A -85,B 0,C 180,E1 -1784.472,E2 -1784.472} C_VEL
LIN {X 0,Y 580.836,Z 292.296,A -85,B 0,C 180,E1 -1785.628,E2 -1785.628} C_VEL
LIN {X 0,Y 580.28,Z 288.813,A -85,B 0,C 180,E1 -1785.701,E2 -1785.701} C_VEL
LIN {X 0,Y 580.33,Z 274.246,A -85,B 0,C 180,E1 -1788.474,E2 -1788.474} C_VEL
LIN {X 0,Y 580.264,Z 268.202,A -85,B 0,C 180,E1 -1789.665,E2 -1789.665} C_VEL
LIN {X 0,Y 580.28,Z 268.2,A -85,B 0,C 180,E1 -1792.344,E2 -1792.344} C_VEL
LIN {X 0,Y 580.286,Z 268.203,A -85,B 0,C 180,E1 -1795.137,E2 -1795.137} C_VEL
LIN {X 0,Y 580.267,Z 268.199,A -85,B 0,C 180,E1 -1797.918,E2 -1797.918} C_VEL
LIN {X 0,Y 580.319,Z 268.199,A -85,B 0,C 180,E1 -1800.694,E2 -1800.694} C_VEL
LIN {X 0,Y 580.245,Z 268.204,A -85,B 0,C 180,E1 -1803.472,E2 -1803.472} C_VEL
LIN {X 0,Y 580.278,Z 268.199,A -85,B 0,C 180,E1 -1805.561,E2 -1805.561} C_VEL
LIN {X 0,Y 580.276,Z 268.199,A -85,B 0,C 180,E1 -1808.357,E2 -1808.357} C_VEL
LIN {X 0,Y 580.319,Z 268.199,A -85,B 0,C 180,E1 -1811.235,E2 -1811.235} C_VEL
LIN {X 0,Y 580.254,Z 268.201,A -85,B 0,C 180,E1 -1814.341,E2 -1814.341} C_VEL
LIN {X 0,Y 580.256,Z 268.208,A -85,B 0,C 180,E1 -1816.918,E2 -1816.918} C_VEL
LIN {X 0,Y 580.256,Z 268.2,A -85,B 0,C 180,E1 -1819.824,E2 -1819.824} C_VEL
LIN {X 0,Y 580.227,Z 268.203,A -85,B 0,C 180,E1 -1822.055,E2 -1822.055} C_VEL
LIN {X 0,Y 580.259,Z 268.21,A -85,B 0,C 180,E1 -1825.082,E2 -1825.082} C_VEL
LIN {X 0,Y 580.27,Z 268.199,A -85,B 0,C 180,E1 -1827.867,E2 -1827.867} C_VEL
LIN {X 0,Y 580.246,Z 268.204,A -85,B 0,C 180,E1 -1830.7,E2 -1830.7} C_VEL
LIN {X 0,Y 580.262,Z 268.207,A -85,B 0,C 180,E1 -1833.321,E2 -1833.321} C_VEL
LIN {X 0,Y 580.254,Z 268.202,A -85,B 0,C 180,E1 -1835.767,E2 -1835.767} C_VEL
LIN {X 0,Y 580.247,Z 268.201,A -85,B 0,C 180,E1 -1838.15,E2 -1838.15} C_VEL
LIN {X 0,Y 580.28,Z 268.201,A -85,B 0,C 180,E1 -1840.845,E2 -1840.845} C_VEL
LIN {X 0,Y 580.246,Z 268.205,A -85,B 0,C 180,E1 -1843.661,E2 -1843.661} C_VEL
LIN {X 0,Y 580.252,Z 268.202,A -85,B 0,C 180,E1 -1846.612,E2 -1846.612} C_VEL
LIN {X 0,Y 580.272,Z 268.206,A -85,B 0,C 180,E1 -1849.161,E2 -1849.161} C_VEL
LIN {X 0,Y 580.262,Z 268.201,A -85,B 0,C 180,E1 -1851.931,E2 -1851.931} C_VEL
LIN {X 0,Y 580.228,Z 268.204,A -85,B 0,C 180,E1 -1854.457,E2 -1854.457} C_VEL
LIN {X 0,Y 580.271,Z 268.204,A -85,B 0,C 180,E1 -1856.979,E2 -1856.979} C_VEL
LIN {X 0,Y 580.275,Z 268.208,A -85,B 0,C 180,E1 -1859.429,E2 -1859.429} C_VEL
LIN {X 0,Y 580.245,Z 268.203,A -85,B 0,C 180,E1 -1862.152,E2 -1862.152} C_VEL
LIN {X 0,Y 580.285,Z 268.201,A -85,B 0,C 180,E1 -1864.923,E2 -1864.923} C_VEL
LIN {X 0,Y 580.332,Z 268.36,A -85,B 0,C 180,E1 -1865.903,E2 -1865.903} C_VEL
LIN {X 0,Y 581.031,Z 272.593,A -85,B 0,C 180,E1 -1866.478,E2 -1866.478} C_VEL
LIN {X 0,Y 580.881,Z 291.875,A -85,B 0,C 180,E1 -1869.092,E2 -1869.092} C_VEL
LIN {X 0,Y 580.629,Z 313.709,A -85,B 0,C 180,E1 -1872.025,E2 -1872.025} C_VEL
LIN {X 0,Y 580.502,Z 332.813,A -85,B 0,C 180,E1 -1874.556,E2 -1874.556} C_VEL
LIN {X 0,Y 580.405,Z 346.452,A -85,B 0,C 180,E1 -1876.334,E2 -1876.334} C_VEL
LIN {X 0,Y 580.923,Z 350.923,A -85,B 0,C 180,E1 -1876.402,E2 -1876.402} C_VEL
LIN {X 0,Y 580.797,Z 455.07,A -85,B 0,C 180,E1 -1877.71,E2 -1877.71} C_VEL
LIN {X 0,Y 580.727,Z 468.301,A -85,B 0,C 180,E1 -1878.019,E2 -1878.019} C_VEL
LIN {X 0,Y 580.642,Z 481.162,A -85,B 0,C 180,E1 -1878.467,E2 -1878.467} C_VEL
LIN {X 0,Y 580.563,Z 492.669,A -85,B 0,C 180,E1 -1879.011,E2 -1879.011} C_VEL
LIN {X 0,Y 580.447,Z 504.235,A -85,B 0,C 180,E1 -1879.714,E2 -1879.714} C_VEL
LIN {X 0,Y 580.343,Z 514.625,A -85,B 0,C 180,E1 -1880.505,E2 -1880.505} C_VEL
LIN {X 0,Y 580.27,Z 523.133,A -85,B 0,C 180,E1 -1881.294,E2 -1881.294} C_VEL
LIN {X 0,Y 580.22,Z 530.976,A -85,B 0,C 180,E1 -1882.17,E2 -1882.17} C_VEL
LIN {X 0,Y 580.153,Z 538.659,A -85,B 0,C 180,E1 -1883.223,E2 -1883.223} C_VEL
LIN {X 0,Y 580.139,Z 545.689,A -85,B 0,C 180,E1 -1884.44,E2 -1884.44} C_VEL
LIN {X 0,Y 580.108,Z 550.378,A -85,B 0,C 180,E1 -1885.485,E2 -1885.485} C_VEL
LIN {X 0,Y 580.122,Z 553.961,A -85,B 0,C 180,E1 -1886.529,E2 -1886.529} C_VEL
LIN {X 0,Y 580.043,Z 555.812,A -85,B 0,C 180,E1 -1887.223,E2 -1887.223} C_VEL
LIN {X 0,Y 580.039,Z 557.201,A -85,B 0,C 180,E1 -1887.918,E2 -1887.918} C_VEL
LIN {X 0,Y 580.04,Z 558.786,A -85,B 0,C 180,E1 -1889.307,E2 -1889.307} C_VEL
LIN {X 0,Y 580.037,Z 559,A -85,B 0,C 180,E1 -1890.001,E2 -1890.001} C_VEL
LIN {X 0,Y 580.046,Z 558.185,A -85,B 0,C 180,E1 -1891.39,E2 -1891.39} C_VEL
LIN {X 0,Y 580.039,Z 557.199,A -85,B 0,C 180,E1 -1892.084,E2 -1892.084} C_VEL
LIN {X 0,Y 580.043,Z 555.808,A -85,B 0,C 180,E1 -1892.779,E2 -1892.779} C_VEL
LIN {X 0,Y 580.11,Z 552.894,A -85,B 0,C 180,E1 -1893.821,E2 -1893.821} C_VEL
LIN {X 0,Y 580.053,Z 548.947,A -85,B 0,C 180,E1 -1894.866,E2 -1894.866} C_VEL
LIN {X 0,Y 580.139,Z 542.874,A -85,B 0,C 180,E1 -1896.085,E2 -1896.085} C_VEL
LIN {X 0,Y 580.185,Z 536.235,A -85,B 0,C 180,E1 -1897.133,E2 -1897.133} C_VEL
LIN {X 0,Y 580.251,Z 527.988,A -85,B 0,C 180,E1 -1898.182,E2 -1898.182} C_VEL
LIN {X 0,Y 580.308,Z 519.536,A -85,B 0,C 180,E1 -1899.059,E2 -1899.059} C_VEL
LIN {X 0,Y 580.419,Z 509.096,A -85,B 0,C 180,E1 -1899.936,E2 -1899.936} C_VEL
LIN {X 0,Y 580.513,Z 498.755,A -85,B 0,C 180,E1 -1900.639,E2 -1900.639} C_VEL
LIN {X 0,Y 580.581,Z 487.413,A -85,B 0,C 180,E1 -1901.256,E2 -1901.256} C_VEL
LIN {X 0,Y 580.64,Z 475.769,A -85,B 0,C 180,E1 -1901.741,E2 -1901.741} C_VEL
LIN {X 0,Y 580.738,Z 462.353,A -85,B 0,C 180,E1 -1902.138,E2 -1902.138} C_VEL
LIN {X 0,Y 580.819,Z 449.094,A -85,B 0,C 180,E1 -1902.38,E2 -1902.38} C_VEL
LIN {X 0,Y 580.805,Z 349.177,A -85,B 0,C 180,E1 -1903.623,E2 -1903.623} C_VEL
LIN {X 0,Y 580.412,Z 346.271,A -85,B 0,C 180,E1 -1903.68,E2 -1903.68} C_VEL
LIN {X 0,Y 580.607,Z 323.244,A -85,B 0,C 180,E1 -1906.707,E2 -1906.707} C_VEL
LIN {X 0,Y 580.796,Z 300.045,A -85,B 0,C 180,E1 -1909.804,E2 -1909.804} C_VEL
LIN {X 0,Y 581.066,Z 278.211,A -85,B 0,C 180,E1 -1912.769,E2 -1912.769} C_VEL
LIN {X 0,Y 580.88,Z 271.25,A -85,B 0,C 180,E1 -1913.72,E2 -1913.72} C_VEL
LIN {X 0,Y 580.292,Z 268.204,A -85,B 0,C 180,E1 -1914.173,E2 -1914.173} C_VEL
LIN {X 0,Y 580.234,Z 268.213,A -85,B 0,C 180,E1 -1916.624,E2 -1916.624} C_VEL
LIN {X 0,Y 580.268,Z 268.199,A -85,B 0,C 180,E1 -1919.303,E2 -1919.303} C_VEL
LIN {X 0,Y 580.289,Z 268.2,A -85,B 0,C 180,E1 -1922.199,E2 -1922.199} C_VEL
LIN {X 0,Y 580.269,Z 268.208,A -85,B 0,C 180,E1 -1924.695,E2 -1924.695} C_VEL
LIN {X 0,Y 580.256,Z 268.201,A -85,B 0,C 180,E1 -1927.269,E2 -1927.269} C_VEL
LIN {X 0,Y 580.269,Z 268.202,A -85,B 0,C 180,E1 -1930.267,E2 -1930.267} C_VEL
LIN {X 0,Y 580.254,Z 268.21,A -85,B 0,C 180,E1 -1932.705,E2 -1932.705} C_VEL
LIN {X 0,Y 580.234,Z 268.202,A -85,B 0,C 180,E1 -1935.608,E2 -1935.608} C_VEL
LIN {X 0,Y 580.251,Z 268.211,A -85,B 0,C 180,E1 -1938.667,E2 -1938.667} C_VEL
LIN {X 0,Y 580.241,Z 268.207,A -85,B 0,C 180,E1 -1940.962,E2 -1940.962} C_VEL
LIN {X 0,Y 580.219,Z 268.205,A -85,B 0,C 180,E1 -1943.592,E2 -1943.592} C_VEL
LIN {X 0,Y 580.246,Z 268.203,A -85,B 0,C 180,E1 -1946.14,E2 -1946.14} C_VEL
LIN {X 0,Y 580.247,Z 268.21,A -85,B 0,C 180,E1 -1948.612,E2 -1948.612} C_VEL
LIN {X 0,Y 580.249,Z 268.206,A -85,B 0,C 180,E1 -1951.021,E2 -1951.021} C_VEL
LIN {X 0,Y 580.231,Z 268.203,A -85,B 0,C 180,E1 -1953.669,E2 -1953.669} C_VEL
LIN {X 0,Y 580.222,Z 268.21,A -85,B 0,C 180,E1 -1956.439,E2 -1956.439} C_VEL
LIN {X 0,Y 580.228,Z 268.204,A -85,B 0,C 180,E1 -1959.435,E2 -1959.435} C_VEL
LIN {X 0,Y 580.218,Z 268.205,A -85,B 0,C 180,E1 -1961.643,E2 -1961.643} C_VEL
LIN {X 0,Y 580.233,Z 268.203,A -85,B 0,C 180,E1 -1963.824,E2 -1963.824} C_VEL
LIN {X 0,Y 580.238,Z 268.212,A -85,B 0,C 180,E1 -1966.695,E2 -1966.695} C_VEL
LIN {X 0,Y 580.271,Z 268.199,A -85,B 0,C 180,E1 -1969.532,E2 -1969.532} C_VEL
LIN {X 0,Y 580.294,Z 268.199,A -85,B 0,C 180,E1 -1972.344,E2 -1972.344} C_VEL
LIN {X 0,Y 580.298,Z 268.199,A -85,B 0,C 180,E1 -1975.136,E2 -1975.136} C_VEL
LIN {X 0,Y 580.283,Z 268.197,A -85,B 0,C 180,E1 -1977.917,E2 -1977.917} C_VEL
LIN {X 0,Y 580.339,Z 268.199,A -85,B 0,C 180,E1 -1980.694,E2 -1980.694} C_VEL
LIN {X 0,Y 580.253,Z 268.202,A -85,B 0,C 180,E1 -1983.472,E2 -1983.472} C_VEL
LIN {X 0,Y 580.289,Z 268.197,A -85,B 0,C 180,E1 -1985.56,E2 -1985.56} C_VEL
LIN {X 0,Y 580.294,Z 268.199,A -85,B 0,C 180,E1 -1988.356,E2 -1988.356} C_VEL
LIN {X 0,Y 580.34,Z 268.194,A -85,B 0,C 180,E1 -1991.234,E2 -1991.234} C_VEL
LIN {X 0,Y 580.273,Z 268.201,A -85,B 0,C 180,E1 -1994.34,E2 -1994.34} C_VEL
LIN {X 0,Y 580.275,Z 268.208,A -85,B 0,C 180,E1 -1996.916,E2 -1996.916} C_VEL
LIN {X 0,Y 580.274,Z 268.198,A -85,B 0,C 180,E1 -1999.823,E2 -1999.823} C_VEL
LIN {X 0,Y 580.251,Z 268.204,A -85,B 0,C 180,E1 -2001.358,E2 -2001.358} C_VEL
LIN {X 0,Y 579.556,Z 268.29,A -85,B 0,C 180,E1 -2001.937,E2 -2001.937} C_VEL
LIN {X 0,Y 576.678,Z 268.655,A -85,B 0,C 180,E1 -2002.877,E2 -2002.877} C_VEL
LIN {X 0,Y 574.281,Z 268.949,A -85,B 0,C 180,E1 -2003.633,E2 -2003.633} C_VEL
LIN {X 0,Y 573.282,Z 269.071,A -85,B 0,C 180,E1 -2004.217,E2 -2004.217} C_VEL
LIN {X 0,Y 573.216,Z 269.081,A -85,B 0,C 180,E1 -2004.415,E2 -2004.415} C_VEL
LIN {X 0,Y 573.236,Z 269.084,A -85,B 0,C 180,E1 -2006.976,E2 -2006.976} C_VEL
LIN {X 0,Y 573.222,Z 269.078,A -85,B 0,C 180,E1 -2009.492,E2 -2009.492} C_VEL
LIN {X 0,Y 573.224,Z 269.077,A -85,B 0,C 180,E1 -2012.231,E2 -2012.231} C_VEL
LIN {X 0,Y 573.226,Z 269.084,A -85,B 0,C 180,E1 -2014.776,E2 -2014.776} C_VEL
LIN {X 0,Y 573.228,Z 269.082,A -85,B 0,C 180,E1 -2017.168,E2 -2017.168} C_VEL
LIN {X 0,Y 573.224,Z 269.077,A -85,B 0,C 180,E1 -2019.608,E2 -2019.608} C_VEL
LIN {X 0,Y 573.217,Z 269.08,A -85,B 0,C 180,E1 -2022.402,E2 -2022.402} C_VEL
LIN {X 0,Y 573.204,Z 269.085,A -85,B 0,C 180,E1 -2024.677,E2 -2024.677} C_VEL
LIN {X 0,Y 573.231,Z 269.079,A -85,B 0,C 180,E1 -2027.359,E2 -2027.359} C_VEL
LIN {X 0,Y 573.255,Z 269.075,A -85,B 0,C 180,E1 -2029.479,E2 -2029.479} C_VEL
LIN {X 0,Y 573.221,Z 269.077,A -85,B 0,C 180,E1 -2032.194,E2 -2032.194} C_VEL
LIN {X 0,Y 573.253,Z 269.08,A -85,B 0,C 180,E1 -2034.818,E2 -2034.818} C_VEL
LIN {X 0,Y 573.243,Z 269.074,A -85,B 0,C 180,E1 -2037.772,E2 -2037.772} C_VEL
LIN {X 0,Y 573.254,Z 269.077,A -85,B 0,C 180,E1 -2040.636,E2 -2040.636} C_VEL
LIN {X 0,Y 573.243,Z 269.083,A -85,B 0,C 180,E1 -2043.025,E2 -2043.025} C_VEL
LIN {X 0,Y 573.267,Z 269.075,A -85,B 0,C 180,E1 -2045.367,E2 -2045.367} C_VEL
LIN {X 0,Y 573.222,Z 269.078,A -85,B 0,C 180,E1 -2048.42,E2 -2048.42} C_VEL
LIN {X 0,Y 573.273,Z 269.075,A -85,B 0,C 180,E1 -2050.729,E2 -2050.729} C_VEL
LIN {X 0,Y 573.248,Z 269.075,A -85,B 0,C 180,E1 -2053.622,E2 -2053.622} C_VEL
LIN {X 0,Y 573.269,Z 269.071,A -85,B 0,C 180,E1 -2055.807,E2 -2055.807} C_VEL
LIN {X 0,Y 573.26,Z 269.077,A -85,B 0,C 180,E1 -2058.745,E2 -2058.745} C_VEL
LIN {X 0,Y 573.286,Z 269.071,A -85,B 0,C 180,E1 -2061.54,E2 -2061.54} C_VEL
LIN {X 0,Y 573.286,Z 269.069,A -85,B 0,C 180,E1 -2064.371,E2 -2064.371} C_VEL
LIN {X 0,Y 573.312,Z 269.066,A -85,B 0,C 180,E1 -2067.892,E2 -2067.892} C_VEL
LIN {X 0,Y 573.327,Z 269.067,A -85,B 0,C 180,E1 -2070.701,E2 -2070.701} C_VEL
LIN {X 0,Y 573.301,Z 269.072,A -85,B 0,C 180,E1 -2072.809,E2 -2072.809} C_VEL
LIN {X 0,Y 573.294,Z 269.07,A -85,B 0,C 180,E1 -2075.626,E2 -2075.626} C_VEL
LIN {X 0,Y 573.28,Z 269.07,A -85,B 0,C 180,E1 -2078.458,E2 -2078.458} C_VEL
LIN {X 0,Y 573.265,Z 269.078,A -85,B 0,C 180,E1 -2081.31,E2 -2081.31} C_VEL
LIN {X 0,Y 573.266,Z 269.071,A -85,B 0,C 180,E1 -2084.191,E2 -2084.191} C_VEL
LIN {X 0,Y 573.25,Z 269.083,A -85,B 0,C 180,E1 -2087.109,E2 -2087.109} C_VEL
LIN {X 0,Y 573.246,Z 269.073,A -85,B 0,C 180,E1 -2090.074,E2 -2090.074} C_VEL
LIN {X 0,Y 573.257,Z 269.082,A -85,B 0,C 180,E1 -2093.151,E2 -2093.151} C_VEL
LIN {X 0,Y 573.274,Z 269.07,A -85,B 0,C 180,E1 -2096.185,E2 -2096.185} C_VEL
LIN {X 0,Y 573.227,Z 269.077,A -85,B 0,C 180,E1 -2098.561,E2 -2098.561} C_VEL
LIN {X 0,Y 573.224,Z 269.083,A -85,B 0,C 180,E1 -2100.989,E2 -2100.989} C_VEL
LIN {X 0,Y 573.263,Z 269.076,A -85,B 0,C 180,E1 -2103.525,E2 -2103.525} C_VEL
LIN {X 0,Y 573.236,Z 269.074,A -85,B 0,C 180,E1 -2106.044,E2 -2106.044} C_VEL
LIN {X 0,Y 573.226,Z 269.078,A -85,B 0,C 180,E1 -2108.697,E2 -2108.697} C_VEL
LIN {X 0,Y 573.234,Z 269.08,A -85,B 0,C 180,E1 -2111.594,E2 -2111.594} C_VEL
LIN {X 0,Y 573.313,Z 269.14,A -85,B 0,C 180,E1 -2114.414,E2 -2114.414} C_VEL
LIN {X 0,Y 573.277,Z 280.633,A -85,B 0,C 180,E1 -2116.645,E2 -2116.645} C_VEL
LIN {X 0,Y 573.237,Z 288.946,A -85,B 0,C 180,E1 -2118.236,E2 -2118.236} C_VEL
LIN {X 0,Y 574.052,Z 295.07,A -85,B 0,C 180,E1 -2118.333,E2 -2118.333} C_VEL
LIN {X 0,Y 573.877,Z 395.626,A -85,B 0,C 180,E1 -2119.616,E2 -2119.616} C_VEL
LIN {X 0,Y 573.757,Z 409.471,A -85,B 0,C 180,E1 -2119.95,E2 -2119.95} C_VEL
LIN {X 0,Y 573.644,Z 422.428,A -85,B 0,C 180,E1 -2120.426,E2 -2120.426} C_VEL
LIN {X 0,Y 573.521,Z 433.714,A -85,B 0,C 180,E1 -2120.983,E2 -2120.983} C_VEL
LIN {X 0,Y 573.406,Z 443.562,A -85,B 0,C 180,E1 -2121.59,E2 -2121.59} C_VEL
LIN {X 0,Y 573.361,Z 452.845,A -85,B 0,C 180,E1 -2122.288,E2 -2122.288} C_VEL
LIN {X 0,Y 573.244,Z 461.564,A -85,B 0,C 180,E1 -2123.077,E2 -2123.077} C_VEL
LIN {X 0,Y 573.161,Z 470.123,A -85,B 0,C 180,E1 -2124.016,E2 -2124.016} C_VEL
LIN {X 0,Y 573.078,Z 477.796,A -85,B 0,C 180,E1 -2125.049,E2 -2125.049} C_VEL
LIN {X 0,Y 573.032,Z 483.949,A -85,B 0,C 180,E1 -2126.081,E2 -2126.081} C_VEL
LIN {X 0,Y 573.01,Z 488.086,A -85,B 0,C 180,E1 -2126.921,E2 -2126.921} C_VEL
LIN {X 0,Y 572.966,Z 492.829,A -85,B 0,C 180,E1 -2128.168,E2 -2128.168} C_VEL
LIN {X 0,Y 572.968,Z 495.591,A -85,B 0,C 180,E1 -2129.15,E2 -2129.15} C_VEL
LIN {X 0,Y 572.948,Z 496.98,A -85,B 0,C 180,E1 -2129.807,E2 -2129.807} C_VEL
LIN {X 0,Y 572.978,Z 498.148,A -85,B 0,C 180,E1 -2130.619,E2 -2130.619} C_VEL
LIN {X 0,Y 572.916,Z 498.999,A -85,B 0,C 180,E1 -2132.021,E2 -2132.021} C_VEL
LIN {X 0,Y 572.932,Z 498.614,A -85,B 0,C 180,E1 -2133.008,E2 -2133.008} C_VEL
LIN {X 0,Y 572.947,Z 497.732,A -85,B 0,C 180,E1 -2133.795,E2 -2133.795} C_VEL
LIN {X 0,Y 572.976,Z 495.036,A -85,B 0,C 180,E1 -2135.17,E2 -2135.17} C_VEL
LIN {X 0,Y 573.014,Z 490.767,A -85,B 0,C 180,E1 -2136.509,E2 -2136.509} C_VEL
LIN {X 0,Y 573.026,Z 485.749,A -85,B 0,C 180,E1 -2137.654,E2 -2137.654} C_VEL
LIN {X 0,Y 573.084,Z 479.716,A -85,B 0,C 180,E1 -2138.734,E2 -2138.734} C_VEL
LIN {X 0,Y 573.155,Z 472.818,A -85,B 0,C 180,E1 -2139.733,E2 -2139.733} C_VEL
LIN {X 0,Y 573.228,Z 463.612,A -85,B 0,C 180,E1 -2140.81,E2 -2140.81} C_VEL
LIN {X 0,Y 573.348,Z 454.167,A -85,B 0,C 180,E1 -2141.694,E2 -2141.694} C_VEL
LIN {X 0,Y 573.405,Z 444.522,A -85,B 0,C 180,E1 -2142.434,E2 -2142.434} C_VEL
LIN {X 0,Y 573.529,Z 435.666,A -85,B 0,C 180,E1 -2142.996,E2 -2142.996} C_VEL
LIN {X 0,Y 573.615,Z 425.113,A -85,B 0,C 180,E1 -2143.541,E2 -2143.541} C_VEL
LIN {X 0,Y 573.693,Z 413.675,A -85,B 0,C 180,E1 -2144.001,E2 -2144.001} C_VEL
LIN {X 0,Y 573.777,Z 400.928,A -85,B 0,C 180,E1 -2144.368,E2 -2144.368} C_VEL
LIN {X 0,Y 573.866,Z 387.507,A -85,B 0,C 180,E1 -2144.598,E2 -2144.598} C_VEL
LIN {X 0,Y 573.992,Z 293.372,A -85,B 0,C 180,E1 -2145.78,E2 -2145.78} C_VEL
LIN {X 0,Y 573.226,Z 288.802,A -85,B 0,C 180,E1 -2145.874,E2 -2145.874} C_VEL
LIN {X 0,Y 573.346,Z 274.196,A -85,B 0,C 180,E1 -2148.69,E2 -2148.69} C_VEL
LIN {X 0,Y 573.226,Z 269.079,A -85,B 0,C 180,E1 -2149.715,E2 -2149.715} C_VEL
LIN {X 0,Y 573.229,Z 269.078,A -85,B 0,C 180,E1 -2152.25,E2 -2152.25} C_VEL
LIN {X 0,Y 573.258,Z 269.08,A -85,B 0,C 180,E1 -2155.077,E2 -2155.077} C_VEL
LIN {X 0,Y 573.239,Z 269.075,A -85,B 0,C 180,E1 -2157.893,E2 -2157.893} C_VEL
LIN {X 0,Y 573.287,Z 269.075,A -85,B 0,C 180,E1 -2160.703,E2 -2160.703} C_VEL
LIN {X 0,Y 573.195,Z 269.082,A -85,B 0,C 180,E1 -2163.515,E2 -2163.515} C_VEL
LIN {X 0,Y 573.242,Z 269.075,A -85,B 0,C 180,E1 -2165.629,E2 -2165.629} C_VEL
LIN {X 0,Y 573.249,Z 269.075,A -85,B 0,C 180,E1 -2168.46,E2 -2168.46} C_VEL
LIN {X 0,Y 573.263,Z 269.076,A -85,B 0,C 180,E1 -2171.312,E2 -2171.312} C_VEL
LIN {X 0,Y 573.22,Z 269.078,A -85,B 0,C 180,E1 -2174.427,E2 -2174.427} C_VEL
LIN {X 0,Y 573.202,Z 269.087,A -85,B 0,C 180,E1 -2177.114,E2 -2177.114} C_VEL
LIN {X 0,Y 573.205,Z 269.077,A -85,B 0,C 180,E1 -2180.079,E2 -2180.079} C_VEL
LIN {X 0,Y 573.188,Z 269.081,A -85,B 0,C 180,E1 -2182.34,E2 -2182.34} C_VEL
LIN {X 0,Y 573.207,Z 269.083,A -85,B 0,C 180,E1 -2185.413,E2 -2185.413} C_VEL
LIN {X 0,Y 573.214,Z 269.077,A -85,B 0,C 180,E1 -2188.035,E2 -2188.035} C_VEL
LIN {X 0,Y 573.193,Z 269.086,A -85,B 0,C 180,E1 -2190.888,E2 -2190.888} C_VEL
LIN {X 0,Y 573.242,Z 269.078,A -85,B 0,C 180,E1 -2193.532,E2 -2193.532} C_VEL
LIN {X 0,Y 573.209,Z 269.078,A -85,B 0,C 180,E1 -2196.052,E2 -2196.052} C_VEL
LIN {X 0,Y 573.21,Z 269.08,A -85,B 0,C 180,E1 -2198.705,E2 -2198.705} C_VEL
LIN {X 0,Y 573.23,Z 269.079,A -85,B 0,C 180,E1 -2201.601,E2 -2201.601} C_VEL
LIN {X 0,Y 573.197,Z 269.079,A -85,B 0,C 180,E1 -2204.338,E2 -2204.338} C_VEL
LIN {X 0,Y 573.218,Z 269.086,A -85,B 0,C 180,E1 -2207.361,E2 -2207.361} C_VEL
LIN {X 0,Y 573.246,Z 269.08,A -85,B 0,C 180,E1 -2209.481,E2 -2209.481} C_VEL
LIN {X 0,Y 573.208,Z 269.078,A -85,B 0,C 180,E1 -2212.196,E2 -2212.196} C_VEL
LIN {X 0,Y 573.214,Z 269.087,A -85,B 0,C 180,E1 -2215.232,E2 -2215.232} C_VEL
LIN {X 0,Y 573.234,Z 269.08,A -85,B 0,C 180,E1 -2217.775,E2 -2217.775} C_VEL
LIN {X 0,Y 573.246,Z 269.075,A -85,B 0,C 180,E1 -2220.638,E2 -2220.638} C_VEL
LIN {X 0,Y 573.241,Z 269.08,A -85,B 0,C 180,E1 -2223.813,E2 -2223.813} C_VEL
LIN {X 0,Y 573.295,Z 269.19,A -85,B 0,C 180,E1 -2225.805,E2 -2225.805} C_VEL
LIN {X 0,Y 574.039,Z 274.009,A -85,B 0,C 180,E1 -2226.466,E2 -2226.466} C_VEL
LIN {X 0,Y 573.956,Z 293.376,A -85,B 0,C 180,E1 -2229.035,E2 -2229.035} C_VEL
LIN {X 0,Y 573.671,Z 315.073,A -85,B 0,C 180,E1 -2231.984,E2 -2231.984} C_VEL
LIN {X 0,Y 573.512,Z 334.178,A -85,B 0,C 180,E1 -2234.545,E2 -2234.545} C_VEL
LIN {X 0,Y 573.407,Z 346.452,A -85,B 0,C 180,E1 -2236.164,E2 -2236.164} C_VEL
LIN {X 0,Y 574.052,Z 352.712,A -85,B 0,C 180,E1 -2236.258,E2 -2236.258} C_VEL
LIN {X 0,Y 573.884,Z 455.07,A -85,B 0,C 180,E1 -2237.56,E2 -2237.56} C_VEL
LIN {X 0,Y 573.761,Z 467.538,A -85,B 0,C 180,E1 -2237.849,E2 -2237.849} C_VEL
LIN {X 0,Y 573.669,Z 480.434,A -85,B 0,C 180,E1 -2238.296,E2 -2238.296} C_VEL
LIN {X 0,Y 573.599,Z 492.668,A -85,B 0,C 180,E1 -2238.876,E2 -2238.876} C_VEL
LIN {X 0,Y 573.436,Z 504.232,A -85,B 0,C 180,E1 -2239.587,E2 -2239.587} C_VEL
LIN {X 0,Y 573.329,Z 514.626,A -85,B 0,C 180,E1 -2240.388,E2 -2240.388} C_VEL
LIN {X 0,Y 573.24,Z 523.133,A -85,B 0,C 180,E1 -2241.187,E2 -2241.187} C_VEL
LIN {X 0,Y 573.159,Z 530.976,A -85,B 0,C 180,E1 -2242.073,E2 -2242.073} C_VEL
LIN {X 0,Y 573.072,Z 538.59,A -85,B 0,C 180,E1 -2243.128,E2 -2243.128} C_VEL
LIN {X 0,Y 573.07,Z 545.689,A -85,B 0,C 180,E1 -2244.371,E2 -2244.371} C_VEL
LIN {X 0,Y 573.028,Z 550.378,A -85,B 0,C 180,E1 -2245.429,E2 -2245.429} C_VEL
LIN {X 0,Y 573.022,Z 553.962,A -85,B 0,C 180,E1 -2246.486,E2 -2246.486} C_VEL
LIN {X 0,Y 572.959,Z 555.811,A -85,B 0,C 180,E1 -2247.189,E2 -2247.189} C_VEL
LIN {X 0,Y 572.946,Z 558.187,A -85,B 0,C 180,E1 -2248.595,E2 -2248.595} C_VEL
LIN {X 0,Y 572.938,Z 559,A -85,B 0,C 180,E1 -2250.001,E2 -2250.001} C_VEL
LIN {X 0,Y 572.946,Z 558.185,A -85,B 0,C 180,E1 -2251.407,E2 -2251.407} C_VEL
LIN {X 0,Y 572.939,Z 557.198,A -85,B 0,C 180,E1 -2252.11,E2 -2252.11} C_VEL
LIN {X 0,Y 572.959,Z 555.808,A -85,B 0,C 180,E1 -2252.813,E2 -2252.813} C_VEL
LIN {X 0,Y 573.015,Z 552.893,A -85,B 0,C 180,E1 -2253.869,E2 -2253.869} C_VEL
LIN {X 0,Y 572.963,Z 548.946,A -85,B 0,C 180,E1 -2254.926,E2 -2254.926} C_VEL
LIN {X 0,Y 573.065,Z 542.874,A -85,B 0,C 180,E1 -2256.161,E2 -2256.161} C_VEL
LIN {X 0,Y 573.12,Z 536.235,A -85,B 0,C 180,E1 -2257.221,E2 -2257.221} C_VEL
LIN {X 0,Y 573.201,Z 527.988,A -85,B 0,C 180,E1 -2258.284,E2 -2258.284} C_VEL
LIN {X 0,Y 573.287,Z 519.536,A -85,B 0,C 180,E1 -2259.17,E2 -2259.17} C_VEL
LIN {X 0,Y 573.413,Z 509.096,A -85,B 0,C 180,E1 -2260.059,E2 -2260.059} C_VEL
LIN {X 0,Y 573.555,Z 497.402,A -85,B 0,C 180,E1 -2260.855,E2 -2260.855} C_VEL
LIN {X 0,Y 573.653,Z 486.291,A -85,B 0,C 180,E1 -2261.447,E2 -2261.447} C_VEL
LIN {X 0,Y 573.72,Z 473.173,A -85,B 0,C 180,E1 -2261.975,E2 -2261.975} C_VEL
LIN {X 0,Y 573.809,Z 460.523,A -85,B 0,C 180,E1 -2262.332,E2 -2262.332} C_VEL
LIN {X 0,Y 573.877,Z 447.321,A -85,B 0,C 180,E1 -2262.555,E2 -2262.555} C_VEL
